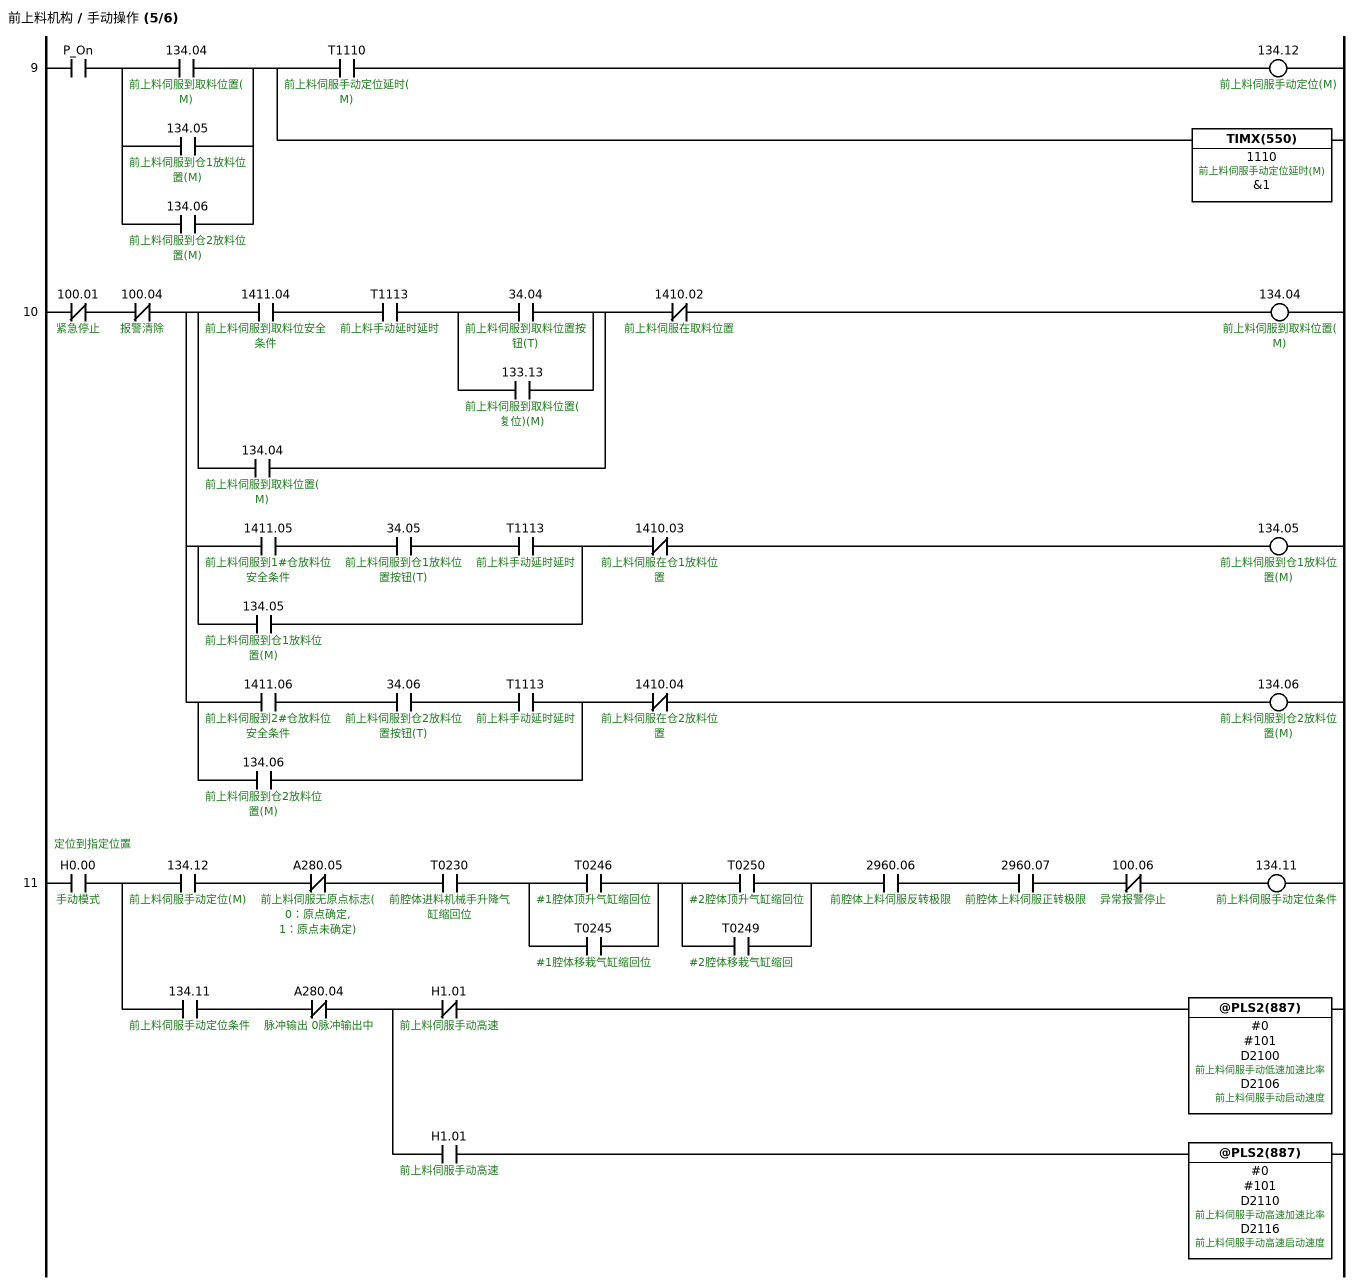
; rung 9
LD P_On
LD 134.04  ; 前上料伺服到取料位置(M)
OR 134.05  ; 前上料伺服到仓1放料位置(M)
OR 134.06  ; 前上料伺服到仓2放料位置(M)
ANDLD
OUT TR0
AND T1110  ; 前上料伺服手动定位延时(M)
OUT 134.12  ; 前上料伺服手动定位(M)
LD TR0
TIMX(550) 1110 &1  ; 前上料伺服手动定位延时(M)
; rung 10
LDNOT 100.01  ; 紧急停止
ANDNOT 100.04  ; 报警清除
OUT TR0
LD 1411.04  ; 前上料伺服到取料位安全条件
AND T1113  ; 前上料手动延时延时
LD 34.04  ; 前上料伺服到取料位置按钮(T)
OR 133.13  ; 前上料伺服到取料位置(复位)(M)
ANDLD
OR 134.04  ; 前上料伺服到取料位置(M)
ANDLD
ANDNOT 1410.02  ; 前上料伺服在取料位置
OUT 134.04  ; 前上料伺服到取料位置(M)
LD TR0
LD 1411.05  ; 前上料伺服到1#仓放料位安全条件
AND 34.05  ; 前上料伺服到仓1放料位置按钮(T)
AND T1113  ; 前上料手动延时延时
OR 134.05  ; 前上料伺服到仓1放料位置(M)
ANDLD
ANDNOT 1410.03  ; 前上料伺服在仓1放料位置
OUT 134.05  ; 前上料伺服到仓1放料位置(M)
LD TR0
LD 1411.06  ; 前上料伺服到2#仓放料位安全条件
AND 34.06  ; 前上料伺服到仓2放料位置按钮(T)
AND T1113  ; 前上料手动延时延时
OR 134.06  ; 前上料伺服到仓2放料位置(M)
ANDLD
ANDNOT 1410.04  ; 前上料伺服在仓2放料位置
OUT 134.06  ; 前上料伺服到仓2放料位置(M)
; rung 11: 定位到指定位置
LD H0.00  ; 手动模式
OUT TR0
AND 134.12  ; 前上料伺服手动定位(M)
ANDNOT A280.05  ; 前上料伺服无原点标志(0：原点确定,1：原点未确定)
AND T0230  ; 前腔体进料机械手升降气缸缩回位
LD T0246  ; #1腔体顶升气缸缩回位
OR T0245  ; #1腔体移栽气缸缩回位
ANDLD
LD T0250  ; #2腔体顶升气缸缩回位
OR T0249  ; #2腔体移栽气缸缩回
ANDLD
AND 2960.06  ; 前腔体上料伺服反转极限
AND 2960.07  ; 前腔体上料伺服正转极限
ANDNOT 100.06  ; 异常报警停止
OUT 134.11  ; 前上料伺服手动定位条件
LD TR0
AND 134.11  ; 前上料伺服手动定位条件
ANDNOT A280.04  ; 脉冲输出 0脉冲输出中
OUT TR0
ANDNOT H1.01  ; 前上料伺服手动高速
@PLS2(887) #0 #101 D2100 D2106  ; 前上料伺服手动低速加速比率, 前上料伺服手动启动速度
LD TR0
AND H1.01  ; 前上料伺服手动高速
@PLS2(887) #0 #101 D2110 D2116  ; 前上料伺服手动高速加速比率, 前上料伺服手动高速启动速度

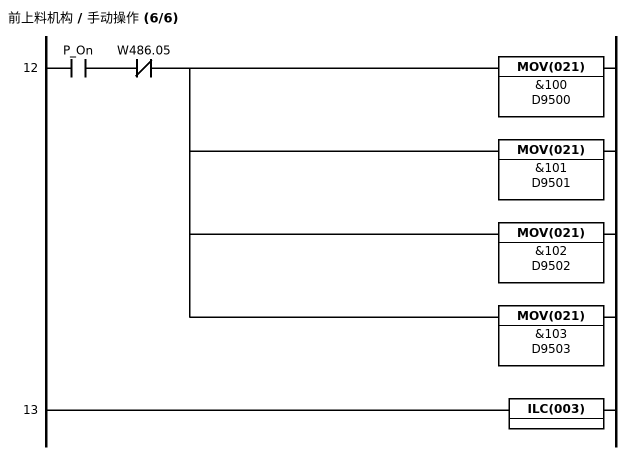
; rung 12
LD P_On
ANDNOT W486.05
MOV(021) &100 D9500
MOV(021) &101 D9501
MOV(021) &102 D9502
MOV(021) &103 D9503
; rung 13
ILC(003)

### Section 自动运行

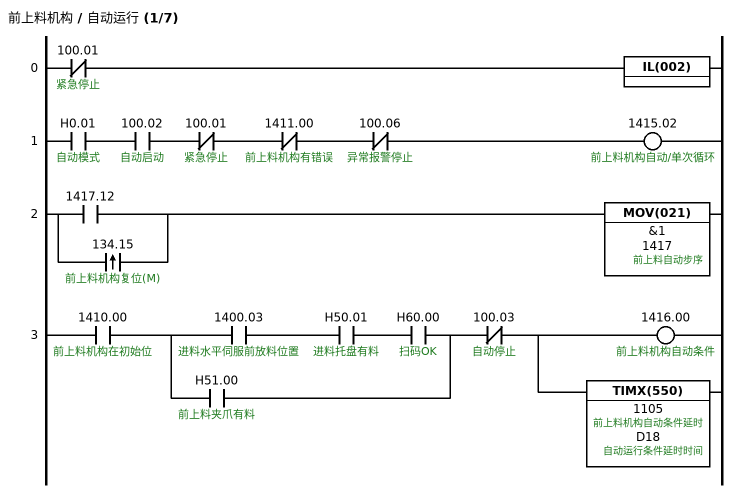
; rung 0
LDNOT 100.01  ; 紧急停止
IL(002)
; rung 1
LD H0.01  ; 自动模式
AND 100.02  ; 自动启动
ANDNOT 100.01  ; 紧急停止
ANDNOT 1411.00  ; 前上料机构有错误
ANDNOT 100.06  ; 异常报警停止
OUT 1415.02  ; 前上料机构自动/单次循环
; rung 2
LD 1417.12
@OR 134.15  ; 前上料机构复位(M)
MOV(021) &1 1417  ; 前上料自动步序
; rung 3
LD 1410.00  ; 前上料机构在初始位
LD 1400.03  ; 进料水平伺服前放料位置
AND H50.01  ; 进料托盘有料
AND H60.00  ; 扫码OK
OR H51.00  ; 前上料夹爪有料
ANDLD
ANDNOT 100.03  ; 自动停止
OUT 1416.00  ; 前上料机构自动条件
TIMX(550) 1105 D18  ; 自动运行条件延时时间, 前上料机构自动条件延时

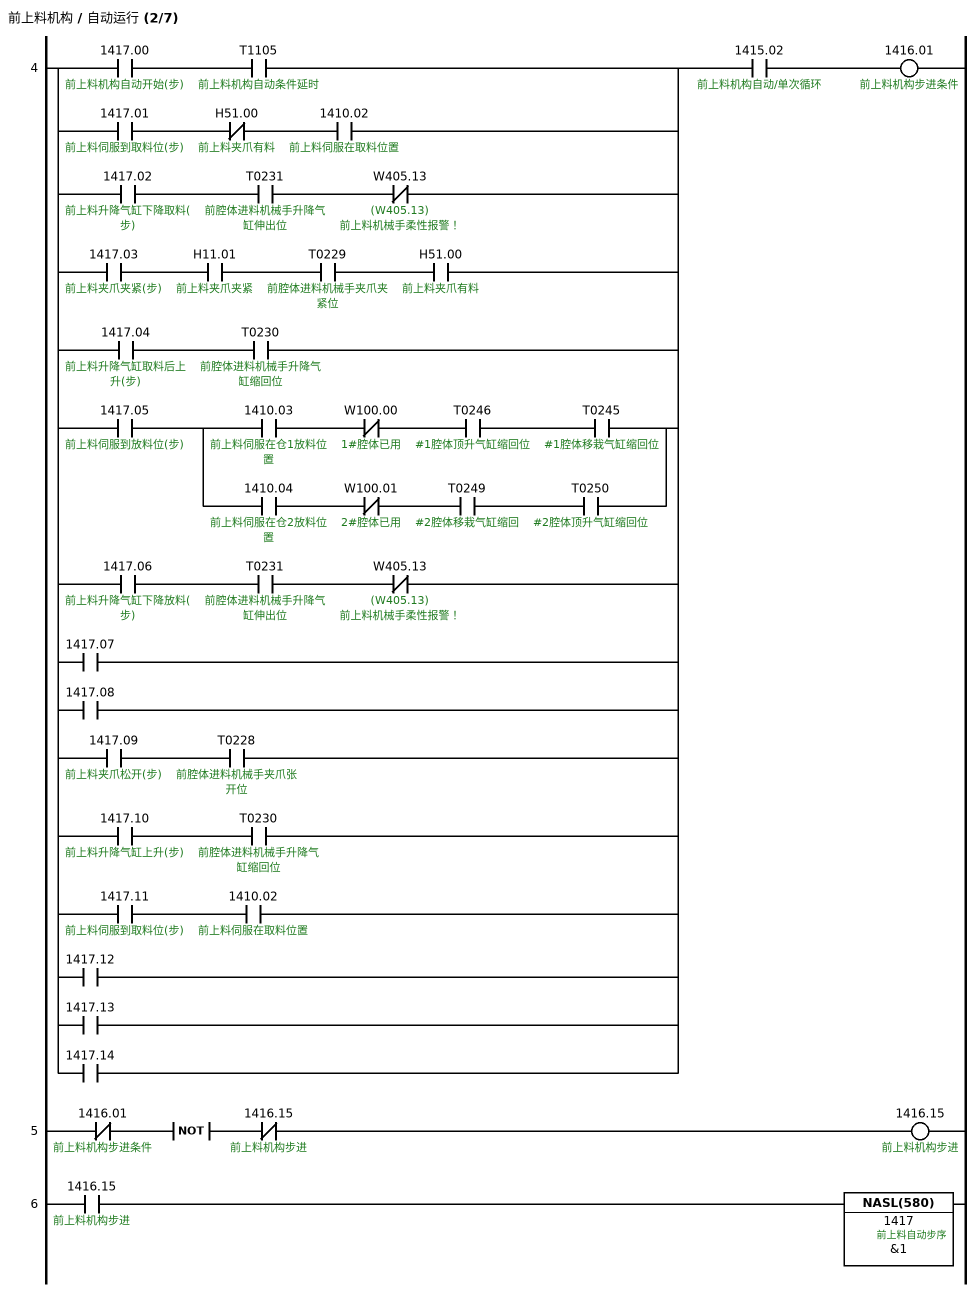
; rung 4
LD 1417.00  ; 前上料机构自动开始(步)
AND T1105  ; 前上料机构自动条件延时
LD 1417.01  ; 前上料伺服到取料位(步)
ANDNOT H51.00  ; 前上料夹爪有料
AND 1410.02  ; 前上料伺服在取料位置
ORLD
LD 1417.02  ; 前上料升降气缸下降取料(步)
AND T0231  ; 前腔体进料机械手升降气缸伸出位
ANDNOT W405.13  ; (W405.13) 前上料机械手柔性报警！
ORLD
LD 1417.03  ; 前上料夹爪夹紧(步)
AND H11.01  ; 前上料夹爪夹紧
AND T0229  ; 前腔体进料机械手夹爪夹紧位
AND H51.00  ; 前上料夹爪有料
ORLD
LD 1417.04  ; 前上料升降气缸取料后上升(步)
AND T0230  ; 前腔体进料机械手升降气缸缩回位
ORLD
LD 1417.05  ; 前上料伺服到放料位(步)
LD 1410.03  ; 前上料伺服在仓1放料位置
ANDNOT W100.00  ; 1#腔体已用
AND T0246  ; #1腔体顶升气缸缩回位
AND T0245  ; #1腔体移栽气缸缩回位
LD 1410.04  ; 前上料伺服在仓2放料位置
ANDNOT W100.01  ; 2#腔体已用
AND T0249  ; #2腔体移栽气缸缩回
AND T0250  ; #2腔体顶升气缸缩回位
ORLD
ANDLD
ORLD
LD 1417.06  ; 前上料升降气缸下降放料(步)
AND T0231  ; 前腔体进料机械手升降气缸伸出位
ANDNOT W405.13  ; (W405.13) 前上料机械手柔性报警！
ORLD
OR 1417.07
OR 1417.08
LD 1417.09  ; 前上料夹爪松开(步)
AND T0228  ; 前腔体进料机械手夹爪张开位
ORLD
LD 1417.10  ; 前上料升降气缸上升(步)
AND T0230  ; 前腔体进料机械手升降气缸缩回位
ORLD
LD 1417.11  ; 前上料伺服到取料位(步)
AND 1410.02  ; 前上料伺服在取料位置
ORLD
OR 1417.12
OR 1417.13
OR 1417.14
AND 1415.02  ; 前上料机构自动/单次循环
OUT 1416.01  ; 前上料机构步进条件
; rung 5
LDNOT 1416.01  ; 前上料机构步进条件
NOT(520)
ANDNOT 1416.15  ; 前上料机构步进
OUT 1416.15  ; 前上料机构步进
; rung 6
LD 1416.15  ; 前上料机构步进
NASL(580) 1417 &1  ; 前上料自动步序

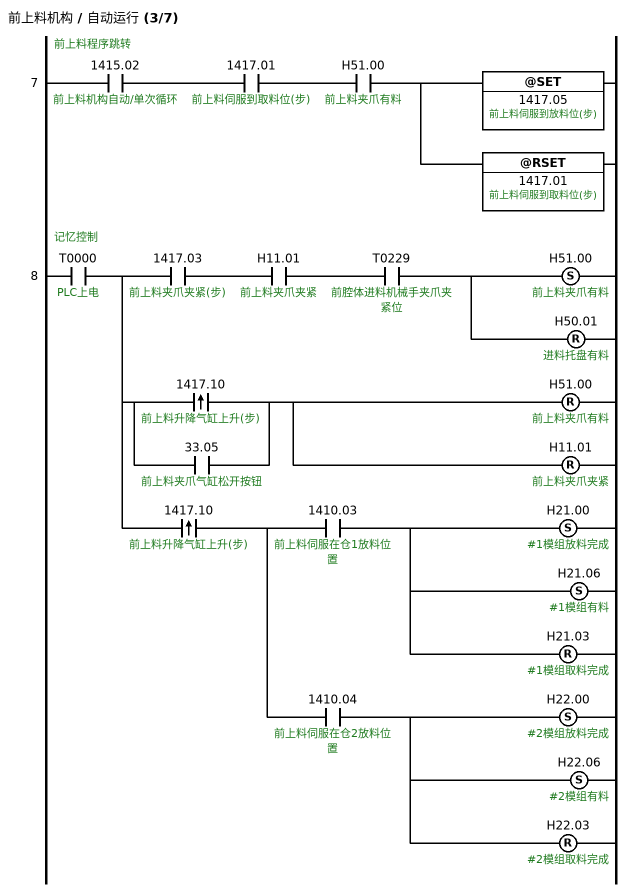
; rung 7: 前上料程序跳转
LD 1415.02  ; 前上料机构自动/单次循环
AND 1417.01  ; 前上料伺服到取料位(步)
AND H51.00  ; 前上料夹爪有料
@SET 1417.05  ; 前上料伺服到放料位(步)
@RSET 1417.01  ; 前上料伺服到取料位(步)
; rung 8: 记忆控制
LD T0000  ; PLC上电
OUT TR0
AND 1417.03  ; 前上料夹爪夹紧(步)
AND H11.01  ; 前上料夹爪夹紧
AND T0229  ; 前腔体进料机械手夹爪夹紧位
SET H51.00  ; 前上料夹爪有料
RSET H50.01  ; 进料托盘有料
LD TR0
@LD 1417.10  ; 前上料升降气缸上升(步)
OR 33.05  ; 前上料夹爪气缸松开按钮
ANDLD
RSET H51.00  ; 前上料夹爪有料
RSET H11.01  ; 前上料夹爪夹紧
LD TR0
@AND 1417.10  ; 前上料升降气缸上升(步)
OUT TR0
AND 1410.03  ; 前上料伺服在仓1放料位置
SET H21.00  ; #1模组放料完成
SET H21.06  ; #1模组有料
RSET H21.03  ; #1模组取料完成
LD TR0
AND 1410.04  ; 前上料伺服在仓2放料位置
SET H22.00  ; #2模组放料完成
SET H22.06  ; #2模组有料
RSET H22.03  ; #2模组取料完成

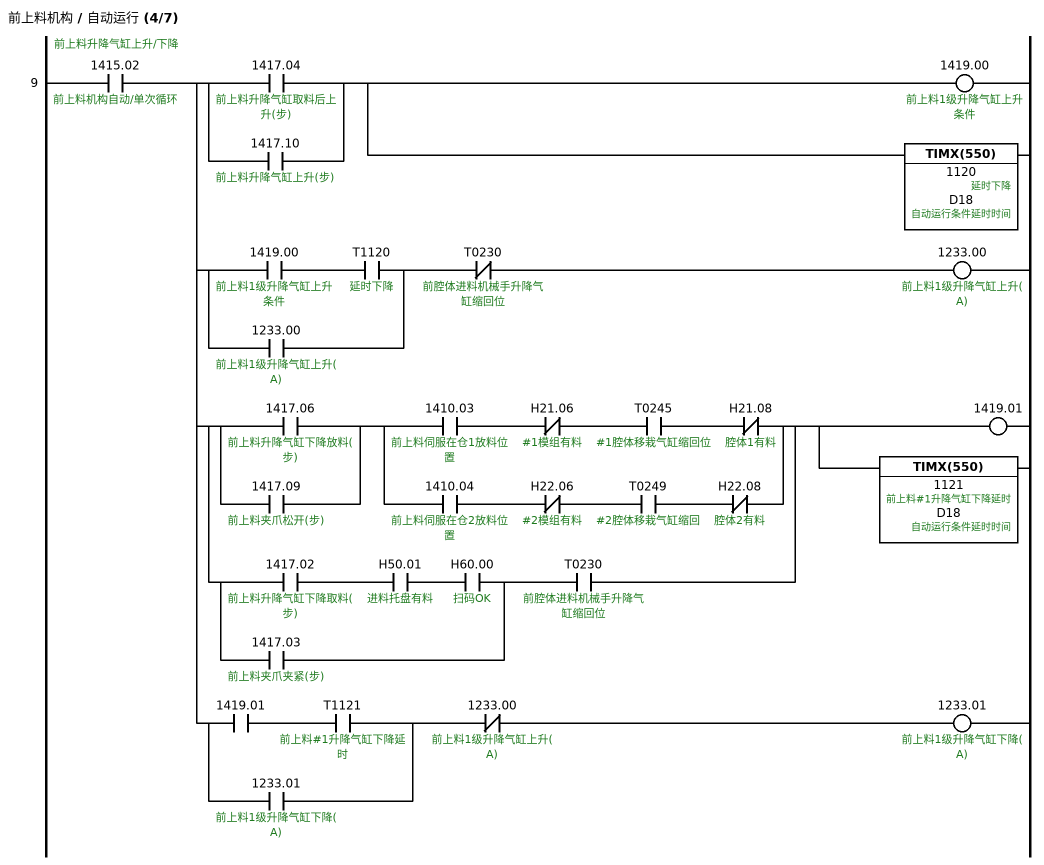
; rung 9: 前上料升降气缸上升/下降
LD 1415.02  ; 前上料机构自动/单次循环
OUT TR0
LD 1417.04  ; 前上料升降气缸取料后上升(步)
OR 1417.10  ; 前上料升降气缸上升(步)
ANDLD
OUT 1419.00  ; 前上料1级升降气缸上升条件
TIMX(550) 1120 D18  ; 自动运行条件延时时间, 延时下降
LD TR0
LD 1419.00  ; 前上料1级升降气缸上升条件
AND T1120  ; 延时下降
OR 1233.00  ; 前上料1级升降气缸上升(A)
ANDLD
ANDNOT T0230  ; 前腔体进料机械手升降气缸缩回位
OUT 1233.00  ; 前上料1级升降气缸上升(A)
LD TR0
LD 1417.06  ; 前上料升降气缸下降放料(步)
OR 1417.09  ; 前上料夹爪松开(步)
LD 1410.03  ; 前上料伺服在仓1放料位置
ANDNOT H21.06  ; #1模组有料
AND T0245  ; #1腔体移栽气缸缩回位
ANDNOT H21.08  ; 腔体1有料
LD 1410.04  ; 前上料伺服在仓2放料位置
ANDNOT H22.06  ; #2模组有料
AND T0249  ; #2腔体移栽气缸缩回
ANDNOT H22.08  ; 腔体2有料
ORLD
ANDLD
LD 1417.02  ; 前上料升降气缸下降取料(步)
AND H50.01  ; 进料托盘有料
AND H60.00  ; 扫码OK
OR 1417.03  ; 前上料夹爪夹紧(步)
AND T0230  ; 前腔体进料机械手升降气缸缩回位
ORLD
ANDLD
OUT 1419.01
TIMX(550) 1121 D18  ; 自动运行条件延时时间, 前上料#1升降气缸下降延时
LD TR0
LD 1419.01
AND T1121  ; 前上料#1升降气缸下降延时
OR 1233.01  ; 前上料1级升降气缸下降(A)
ANDLD
ANDNOT 1233.00  ; 前上料1级升降气缸上升(A)
OUT 1233.01  ; 前上料1级升降气缸下降(A)

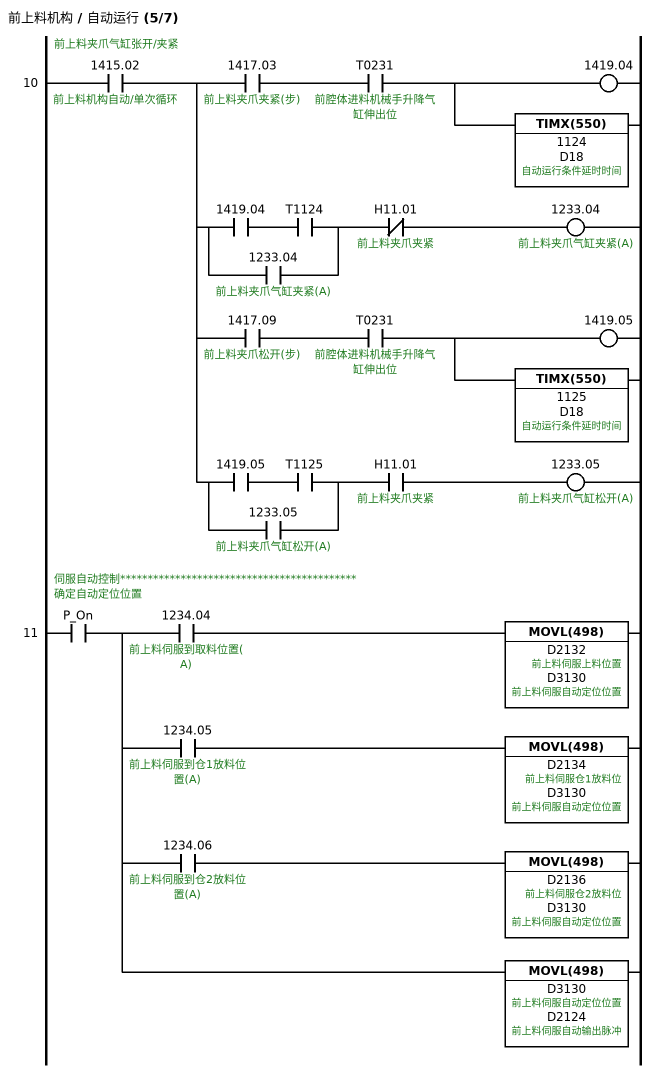
; rung 10: 前上料夹爪气缸张开/夹紧
LD 1415.02  ; 前上料机构自动/单次循环
OUT TR0
AND 1417.03  ; 前上料夹爪夹紧(步)
AND T0231  ; 前腔体进料机械手升降气缸伸出位
OUT 1419.04
TIMX(550) 1124 D18  ; 自动运行条件延时时间
LD TR0
LD 1419.04
AND T1124
OR 1233.04  ; 前上料夹爪气缸夹紧(A)
ANDLD
ANDNOT H11.01  ; 前上料夹爪夹紧
OUT 1233.04  ; 前上料夹爪气缸夹紧(A)
LD TR0
AND 1417.09  ; 前上料夹爪松开(步)
AND T0231  ; 前腔体进料机械手升降气缸伸出位
OUT 1419.05
TIMX(550) 1125 D18  ; 自动运行条件延时时间
LD TR0
LD 1419.05
AND T1125
OR 1233.05  ; 前上料夹爪气缸松开(A)
ANDLD
AND H11.01  ; 前上料夹爪夹紧
OUT 1233.05  ; 前上料夹爪气缸松开(A)
; rung 11: 伺服自动控制******************************************* / 确定自动定位位置
LD P_On
OUT TR0
AND 1234.04  ; 前上料伺服到取料位置(A)
MOVL(498) D2132 D3130  ; 前上料伺服上料位置, 前上料伺服自动定位位置
LD TR0
AND 1234.05  ; 前上料伺服到仓1放料位置(A)
MOVL(498) D2134 D3130  ; 前上料伺服仓1放料位, 前上料伺服自动定位位置
LD TR0
AND 1234.06  ; 前上料伺服到仓2放料位置(A)
MOVL(498) D2136 D3130  ; 前上料伺服仓2放料位, 前上料伺服自动定位位置
LD TR0
MOVL(498) D3130 D2124  ; 前上料伺服自动定位位置, 前上料伺服自动输出脉冲

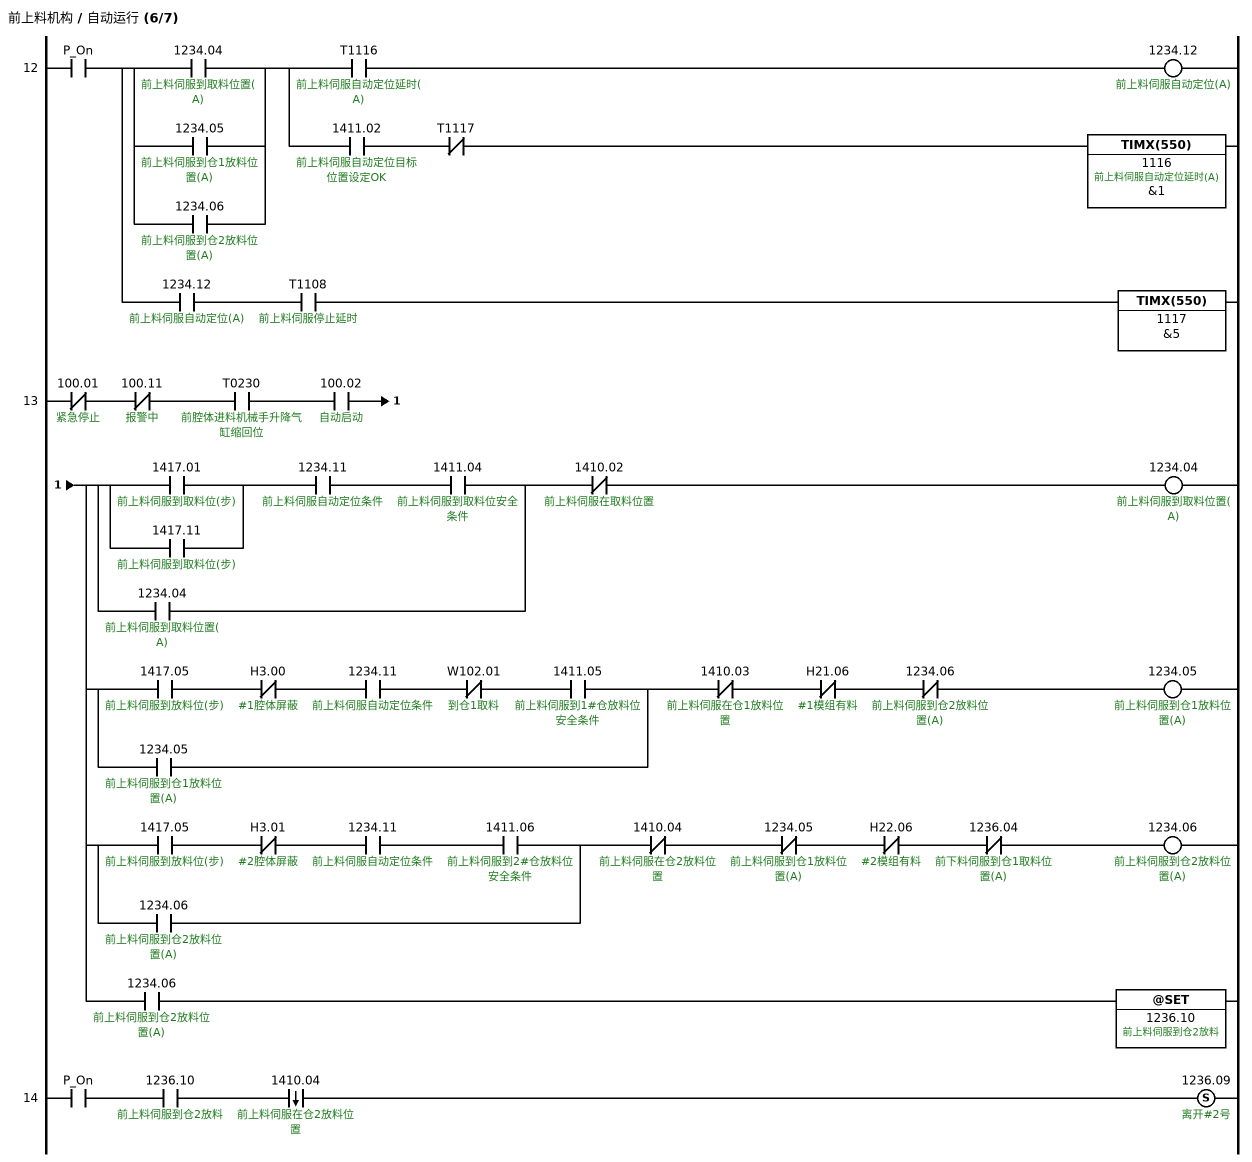
; rung 12
LD P_On
OUT TR0
LD 1234.04  ; 前上料伺服到取料位置(A)
OR 1234.05  ; 前上料伺服到仓1放料位置(A)
OR 1234.06  ; 前上料伺服到仓2放料位置(A)
ANDLD
OUT TR1
AND T1116  ; 前上料伺服自动定位延时(A)
OUT 1234.12  ; 前上料伺服自动定位(A)
LD TR1
AND 1411.02  ; 前上料伺服自动定位目标位置设定OK
ANDNOT T1117
TIMX(550) 1116 &1  ; 前上料伺服自动定位延时(A)
LD TR0
AND 1234.12  ; 前上料伺服自动定位(A)
AND T1108  ; 前上料伺服停止延时
TIMX(550) 1117 &5
; rung 13
LDNOT 100.01  ; 紧急停止
ANDNOT 100.11  ; 报警中
AND T0230  ; 前腔体进料机械手升降气缸缩回位
AND 100.02  ; 自动启动
OUT TR0
LD 1417.01  ; 前上料伺服到取料位(步)
OR 1417.11  ; 前上料伺服到取料位(步)
AND 1234.11  ; 前上料伺服自动定位条件
AND 1411.04  ; 前上料伺服到取料位安全条件
OR 1234.04  ; 前上料伺服到取料位置(A)
ANDLD
ANDNOT 1410.02  ; 前上料伺服在取料位置
OUT 1234.04  ; 前上料伺服到取料位置(A)
LD TR0
LD 1417.05  ; 前上料伺服到放料位(步)
ANDNOT H3.00  ; #1腔体屏蔽
AND 1234.11  ; 前上料伺服自动定位条件
ANDNOT W102.01  ; 到仓1取料
AND 1411.05  ; 前上料伺服到1#仓放料位安全条件
OR 1234.05  ; 前上料伺服到仓1放料位置(A)
ANDLD
ANDNOT 1410.03  ; 前上料伺服在仓1放料位置
ANDNOT H21.06  ; #1模组有料
ANDNOT 1234.06  ; 前上料伺服到仓2放料位置(A)
OUT 1234.05  ; 前上料伺服到仓1放料位置(A)
LD TR0
LD 1417.05  ; 前上料伺服到放料位(步)
ANDNOT H3.01  ; #2腔体屏蔽
AND 1234.11  ; 前上料伺服自动定位条件
AND 1411.06  ; 前上料伺服到2#仓放料位安全条件
OR 1234.06  ; 前上料伺服到仓2放料位置(A)
ANDLD
ANDNOT 1410.04  ; 前上料伺服在仓2放料位置
ANDNOT 1234.05  ; 前上料伺服到仓1放料位置(A)
ANDNOT H22.06  ; #2模组有料
ANDNOT 1236.04  ; 前下料伺服到仓1取料位置(A)
OUT 1234.06  ; 前上料伺服到仓2放料位置(A)
LD TR0
AND 1234.06  ; 前上料伺服到仓2放料位置(A)
@SET 1236.10  ; 前上料伺服到仓2放料
; rung 14
LD P_On
AND 1236.10  ; 前上料伺服到仓2放料
%AND 1410.04  ; 前上料伺服在仓2放料位置
SET 1236.09  ; 离开#2号

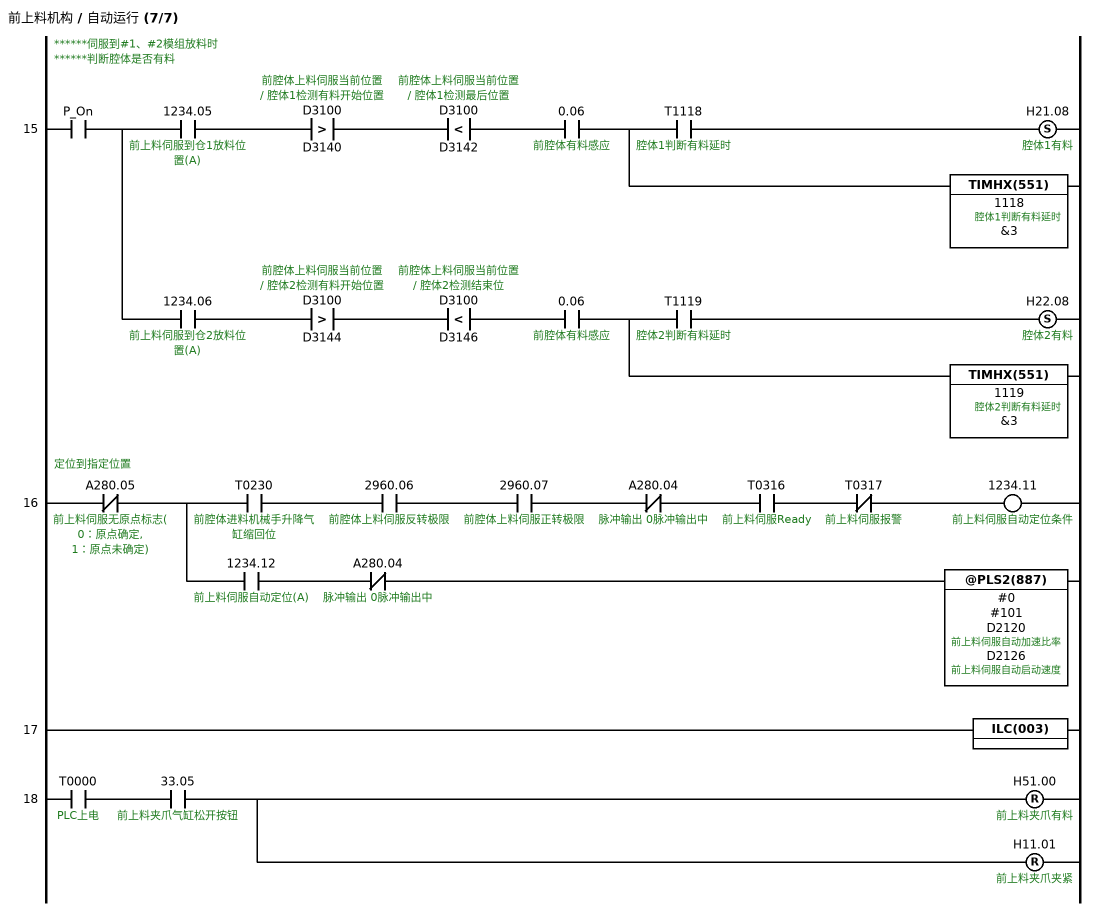
; rung 15: ******伺服到#1、#2模组放料时 / ******判断腔体是否有料
LD P_On
OUT TR0
AND 1234.05  ; 前上料伺服到仓1放料位置(A)
AND>SL(323) D3100 D3140  ; 前腔体上料伺服当前位置, 腔体1检测有料开始位置
AND<SL(313) D3100 D3142  ; 前腔体上料伺服当前位置, 腔体1检测最后位置
AND 0.06  ; 前腔体有料感应
OUT TR1
AND T1118  ; 腔体1判断有料延时
SET H21.08  ; 腔体1有料
LD TR1
TIMHX(551) 1118 &3  ; 腔体1判断有料延时
LD TR0
AND 1234.06  ; 前上料伺服到仓2放料位置(A)
AND>SL(323) D3100 D3144  ; 前腔体上料伺服当前位置, 腔体2检测有料开始位置
AND<SL(313) D3100 D3146  ; 前腔体上料伺服当前位置, 腔体2检测结束位
AND 0.06  ; 前腔体有料感应
OUT TR0
AND T1119  ; 腔体2判断有料延时
SET H22.08  ; 腔体2有料
LD TR0
TIMHX(551) 1119 &3  ; 腔体2判断有料延时
; rung 16: 定位到指定位置
LDNOT A280.05  ; 前上料伺服无原点标志(0：原点确定,1：原点未确定)
OUT TR0
AND T0230  ; 前腔体进料机械手升降气缸缩回位
AND 2960.06  ; 前腔体上料伺服反转极限
AND 2960.07  ; 前腔体上料伺服正转极限
ANDNOT A280.04  ; 脉冲输出 0脉冲输出中
AND T0316  ; 前上料伺服Ready
ANDNOT T0317  ; 前上料伺服报警
OUT 1234.11  ; 前上料伺服自动定位条件
LD TR0
AND 1234.12  ; 前上料伺服自动定位(A)
ANDNOT A280.04  ; 脉冲输出 0脉冲输出中
@PLS2(887) #0 #101 D2120 D2126  ; 前上料伺服自动加速比率, 前上料伺服自动启动速度
; rung 17
ILC(003)
; rung 18
LD T0000  ; PLC上电
AND 33.05  ; 前上料夹爪气缸松开按钮
RSET H51.00  ; 前上料夹爪有料
RSET H11.01  ; 前上料夹爪夹紧

### Section 外部输出

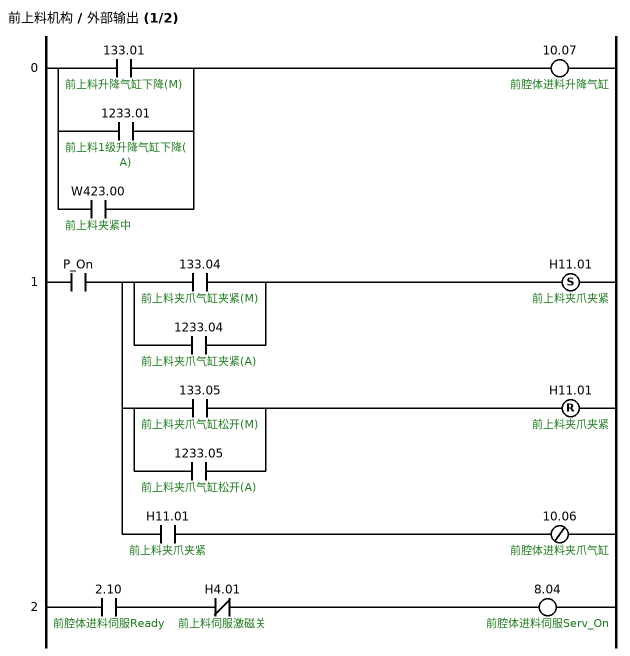
; rung 0
LD 133.01  ; 前上料升降气缸下降(M)
OR 1233.01  ; 前上料1级升降气缸下降(A)
OR W423.00  ; 前上料夹紧中
OUT 10.07  ; 前腔体进料升降气缸
; rung 1
LD P_On
OUT TR0
LD 133.04  ; 前上料夹爪气缸夹紧(M)
OR 1233.04  ; 前上料夹爪气缸夹紧(A)
ANDLD
SET H11.01  ; 前上料夹爪夹紧
LD TR0
LD 133.05  ; 前上料夹爪气缸松开(M)
OR 1233.05  ; 前上料夹爪气缸松开(A)
ANDLD
RSET H11.01  ; 前上料夹爪夹紧
LD TR0
AND H11.01  ; 前上料夹爪夹紧
OUTNOT 10.06  ; 前腔体进料夹爪气缸
; rung 2
LD 2.10  ; 前腔体进料伺服Ready
ANDNOT H4.01  ; 前上料伺服激磁关
OUT 8.04  ; 前腔体进料伺服Serv_On

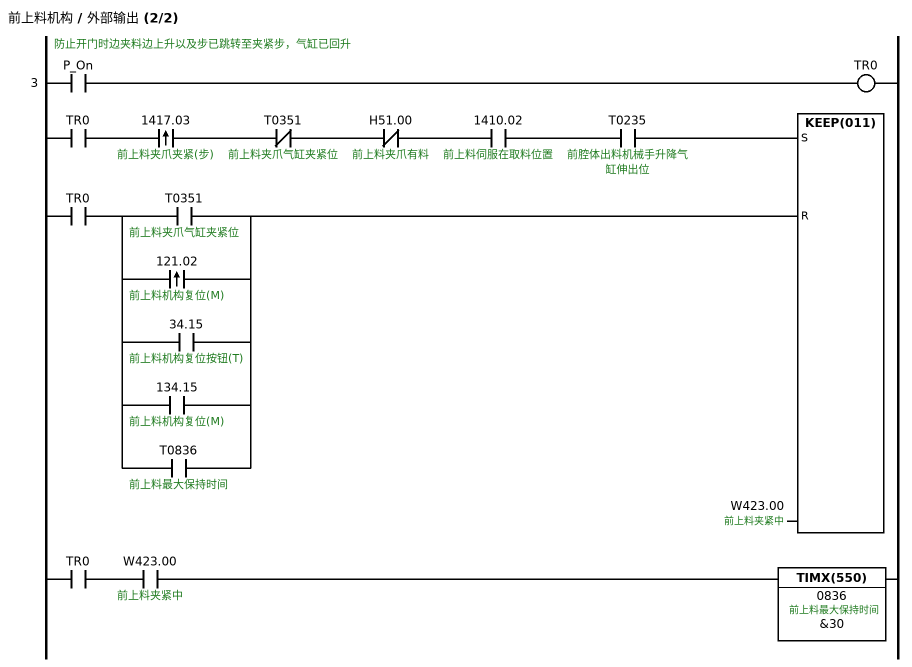
; rung 3: 防止开门时边夹料边上升以及步已跳转至夹紧步，气缸已回升
LD P_On
OUT TR0
@AND 1417.03  ; 前上料夹爪夹紧(步)
ANDNOT T0351  ; 前上料夹爪气缸夹紧位
ANDNOT H51.00  ; 前上料夹爪有料
AND 1410.02  ; 前上料伺服在取料位置
AND T0235  ; 前腔体出料机械手升降气缸伸出位
LD TR0
LD T0351  ; 前上料夹爪气缸夹紧位
@OR 121.02  ; 前上料机构复位(M)
OR 34.15  ; 前上料机构复位按钮(T)
OR 134.15  ; 前上料机构复位(M)
OR T0836  ; 前上料最大保持时间
ANDLD
KEEP(011) W423.00  ; 前上料夹紧中
LD TR0
AND W423.00  ; 前上料夹紧中
TIMX(550) 0836 &30  ; 前上料最大保持时间

### Section 指示灯
; rung 0: ************************************************** / 气缸动作及位置指示灯

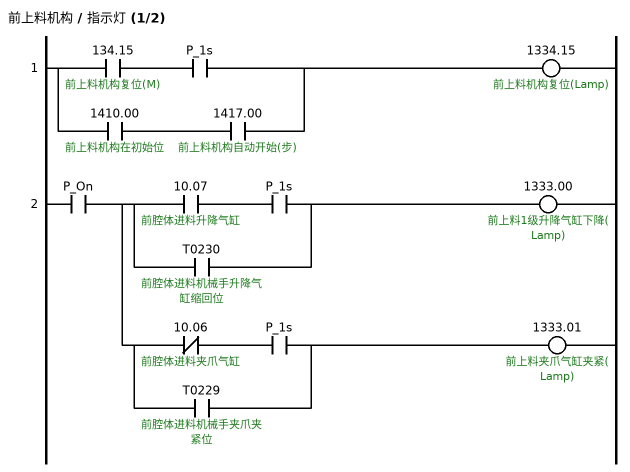
; rung 1
LD 134.15  ; 前上料机构复位(M)
AND P_1s
LD 1410.00  ; 前上料机构在初始位
AND 1417.00  ; 前上料机构自动开始(步)
ORLD
OUT 1334.15  ; 前上料机构复位(Lamp)
; rung 2
LD P_On
OUT TR0
LD 10.07  ; 前腔体进料升降气缸
AND P_1s
OR T0230  ; 前腔体进料机械手升降气缸缩回位
ANDLD
OUT 1333.00  ; 前上料1级升降气缸下降(Lamp)
LD TR0
LDNOT 10.06  ; 前腔体进料夹爪气缸
AND P_1s
OR T0229  ; 前腔体进料机械手夹爪夹紧位
ANDLD
OUT 1333.01  ; 前上料夹爪气缸夹紧(Lamp)

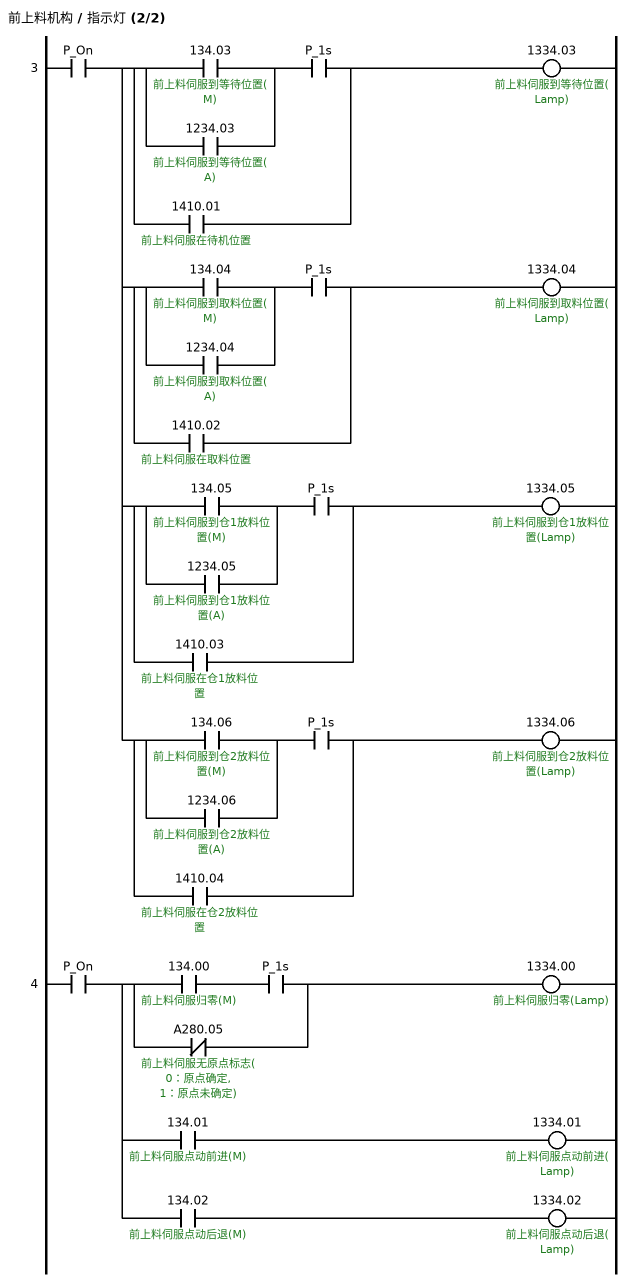
; rung 3
LD P_On
OUT TR0
LD 134.03  ; 前上料伺服到等待位置(M)
OR 1234.03  ; 前上料伺服到等待位置(A)
AND P_1s
OR 1410.01  ; 前上料伺服在待机位置
ANDLD
OUT 1334.03  ; 前上料伺服到等待位置(Lamp)
LD TR0
LD 134.04  ; 前上料伺服到取料位置(M)
OR 1234.04  ; 前上料伺服到取料位置(A)
AND P_1s
OR 1410.02  ; 前上料伺服在取料位置
ANDLD
OUT 1334.04  ; 前上料伺服到取料位置(Lamp)
LD TR0
LD 134.05  ; 前上料伺服到仓1放料位置(M)
OR 1234.05  ; 前上料伺服到仓1放料位置(A)
AND P_1s
OR 1410.03  ; 前上料伺服在仓1放料位置
ANDLD
OUT 1334.05  ; 前上料伺服到仓1放料位置(Lamp)
LD TR0
LD 134.06  ; 前上料伺服到仓2放料位置(M)
OR 1234.06  ; 前上料伺服到仓2放料位置(A)
AND P_1s
OR 1410.04  ; 前上料伺服在仓2放料位置
ANDLD
OUT 1334.06  ; 前上料伺服到仓2放料位置(Lamp)
; rung 4
LD P_On
OUT TR0
LD 134.00  ; 前上料伺服归零(M)
AND P_1s
ORNOT A280.05  ; 前上料伺服无原点标志(0：原点确定,1：原点未确定)
ANDLD
OUT 1334.00  ; 前上料伺服归零(Lamp)
LD TR0
AND 134.01  ; 前上料伺服点动前进(M)
OUT 1334.01  ; 前上料伺服点动前进(Lamp)
LD TR0
AND 134.02  ; 前上料伺服点动后退(M)
OUT 1334.02  ; 前上料伺服点动后退(Lamp)

### Section END
; rung 0
END(001)

## Program 前下料机构 (cyclic task 3)

### Section Main

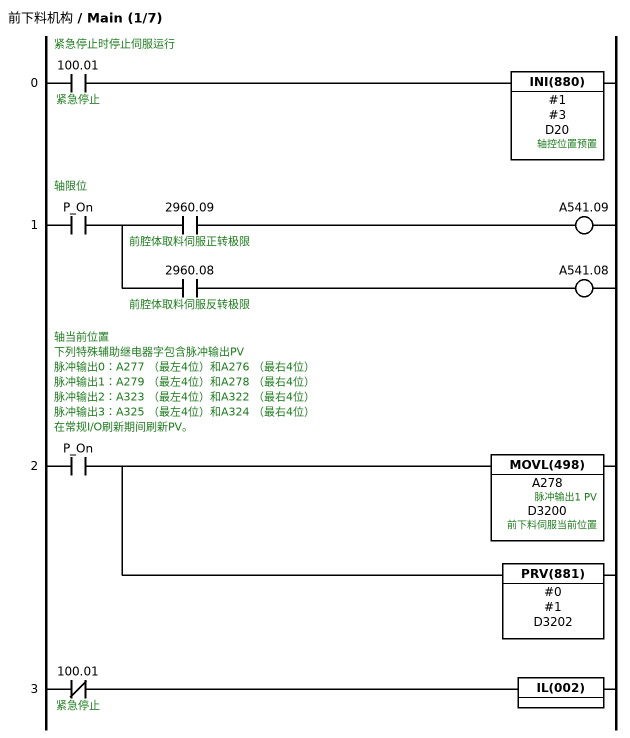
; rung 0: 紧急停止时停止伺服运行
LD 100.01  ; 紧急停止
INI(880) #1 #3 D20  ; 轴控位置预置
; rung 1: 轴限位
LD P_On
OUT TR0
AND 2960.09  ; 前腔体取料伺服正转极限
OUT A541.09
LD TR0
AND 2960.08  ; 前腔体取料伺服反转极限
OUT A541.08
; rung 2: 轴当前位置 / 下列特殊辅助继电器字包含脉冲输出PV / 脉冲输出0：A277 （最左4位）和A276 （最右4位） / 脉冲输出1：A279 （最左4位）和A278 （最右4位） / 脉冲输出2：A323 （最左4位）和A322 （最右4位） / 脉冲输出3：A325 （最左4位）和A324 （最右4位） / 在常规I/O刷新期间刷新PV。
LD P_On
MOVL(498) A278 D3200  ; 脉冲输出1 PV, 前下料伺服当前位置
PRV(881) #0 #1 D3202
; rung 3
LDNOT 100.01  ; 紧急停止
IL(002)

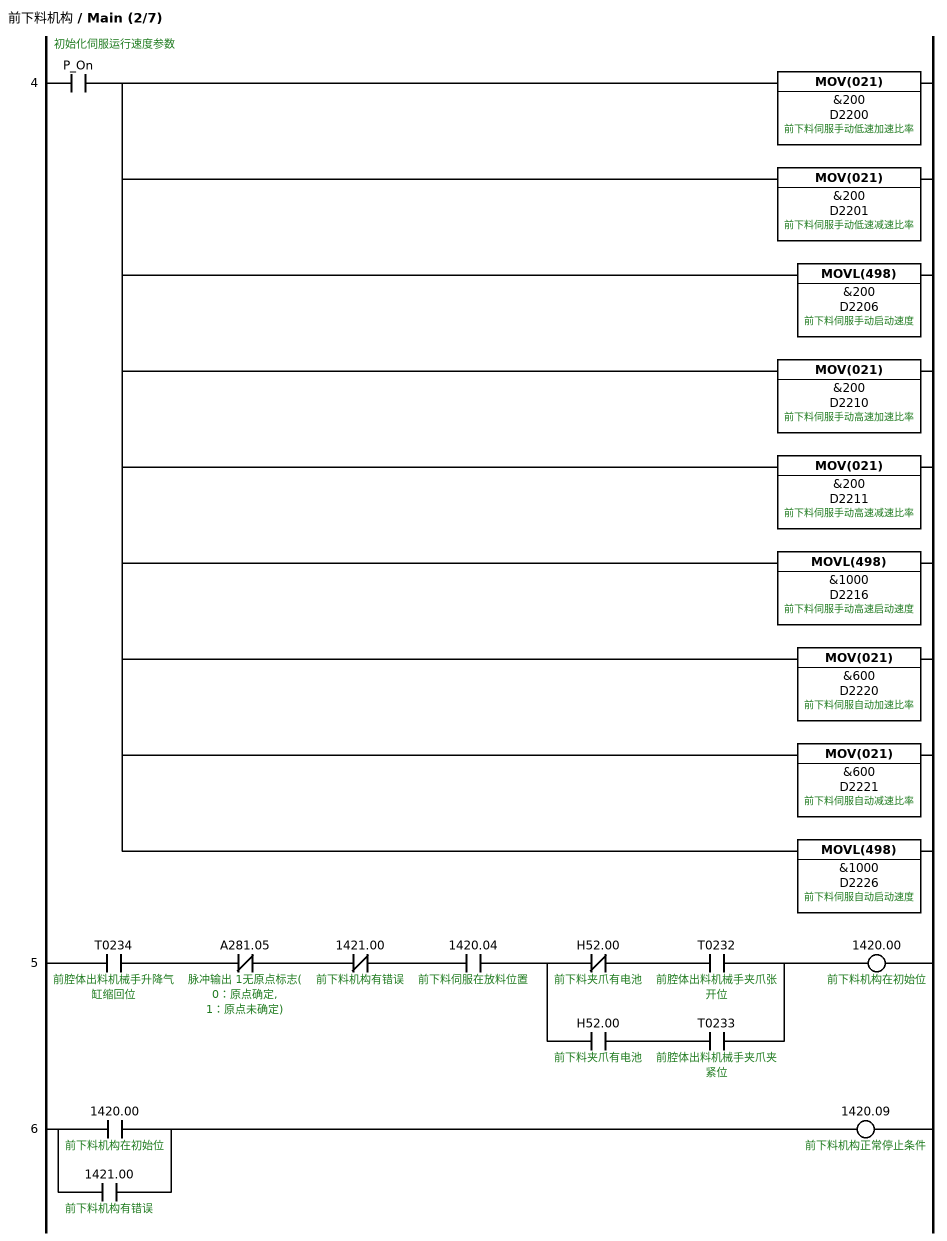
; rung 4: 初始化伺服运行速度参数
LD P_On
MOV(021) &200 D2200  ; 前下料伺服手动低速加速比率
MOV(021) &200 D2201  ; 前下料伺服手动低速减速比率
MOVL(498) &200 D2206  ; 前下料伺服手动启动速度
MOV(021) &200 D2210  ; 前下料伺服手动高速加速比率
MOV(021) &200 D2211  ; 前下料伺服手动高速减速比率
MOVL(498) &1000 D2216  ; 前下料伺服手动高速启动速度
MOV(021) &600 D2220  ; 前下料伺服自动加速比率
MOV(021) &600 D2221  ; 前下料伺服自动减速比率
MOVL(498) &1000 D2226  ; 前下料伺服自动启动速度
; rung 5
LD T0234  ; 前腔体出料机械手升降气缸缩回位
ANDNOT A281.05  ; 脉冲输出 1无原点标志(0：原点确定,1：原点未确定)
ANDNOT 1421.00  ; 前下料机构有错误
AND 1420.04  ; 前下料伺服在放料位置
LDNOT H52.00  ; 前下料夹爪有电池
AND T0232  ; 前腔体出料机械手夹爪张开位
LD H52.00  ; 前下料夹爪有电池
AND T0233  ; 前腔体出料机械手夹爪夹紧位
ORLD
ANDLD
OUT 1420.00  ; 前下料机构在初始位
; rung 6
LD 1420.00  ; 前下料机构在初始位
OR 1421.00  ; 前下料机构有错误
OUT 1420.09  ; 前下料机构正常停止条件

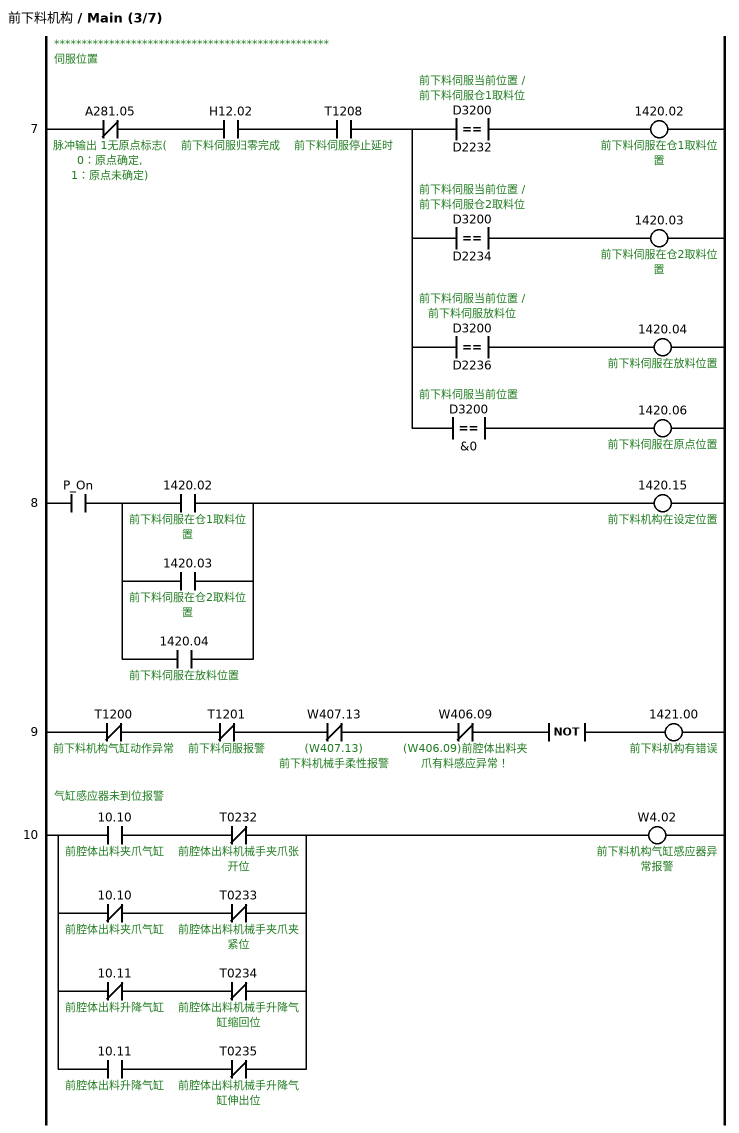
; rung 7: ************************************************** / 伺服位置
LDNOT A281.05  ; 脉冲输出 1无原点标志(0：原点确定,1：原点未确定)
AND H12.02  ; 前下料伺服归零完成
AND T1208  ; 前下料伺服停止延时
OUT TR0
AND=SL(303) D3200 D2232  ; 前下料伺服当前位置, 前下料伺服仓1取料位
OUT 1420.02  ; 前下料伺服在仓1取料位置
LD TR0
AND=SL(303) D3200 D2234  ; 前下料伺服当前位置, 前下料伺服仓2取料位
OUT 1420.03  ; 前下料伺服在仓2取料位置
LD TR0
AND=SL(303) D3200 D2236  ; 前下料伺服当前位置, 前下料伺服放料位
OUT 1420.04  ; 前下料伺服在放料位置
LD TR0
AND=SL(303) D3200 &0  ; 前下料伺服当前位置
OUT 1420.06  ; 前下料伺服在原点位置
; rung 8
LD P_On
LD 1420.02  ; 前下料伺服在仓1取料位置
OR 1420.03  ; 前下料伺服在仓2取料位置
OR 1420.04  ; 前下料伺服在放料位置
ANDLD
OUT 1420.15  ; 前下料机构在设定位置
; rung 9
LDNOT T1200  ; 前下料机构气缸动作异常
ANDNOT T1201  ; 前下料伺服报警
ANDNOT W407.13  ; (W407.13) 前下料机械手柔性报警
ANDNOT W406.09  ; (W406.09)前腔体出料夹爪有料感应异常！
NOT(520)
OUT 1421.00  ; 前下料机构有错误
; rung 10: 气缸感应器未到位报警
LD 10.10  ; 前腔体出料夹爪气缸
ANDNOT T0232  ; 前腔体出料机械手夹爪张开位
LDNOT 10.10  ; 前腔体出料夹爪气缸
ANDNOT T0233  ; 前腔体出料机械手夹爪夹紧位
ORLD
LDNOT 10.11  ; 前腔体出料升降气缸
ANDNOT T0234  ; 前腔体出料机械手升降气缸缩回位
ORLD
LD 10.11  ; 前腔体出料升降气缸
ANDNOT T0235  ; 前腔体出料机械手升降气缸伸出位
ORLD
OUT W4.02  ; 前下料机构气缸感应器异常报警

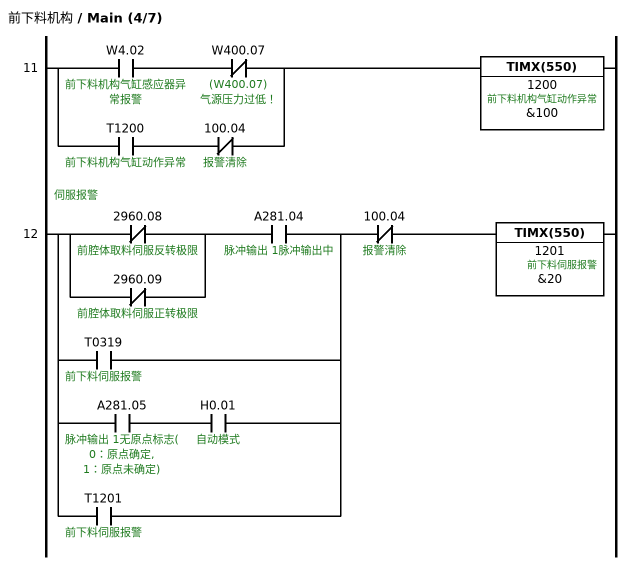
; rung 11
LD W4.02  ; 前下料机构气缸感应器异常报警
ANDNOT W400.07  ; (W400.07) 气源压力过低！
LD T1200  ; 前下料机构气缸动作异常
ANDNOT 100.04  ; 报警清除
ORLD
TIMX(550) 1200 &100  ; 前下料机构气缸动作异常
; rung 12: 伺服报警
LDNOT 2960.08  ; 前腔体取料伺服反转极限
ORNOT 2960.09  ; 前腔体取料伺服正转极限
AND A281.04  ; 脉冲输出 1脉冲输出中
OR T0319  ; 前下料伺服报警
LD A281.05  ; 脉冲输出 1无原点标志(0：原点确定,1：原点未确定)
AND H0.01  ; 自动模式
ORLD
OR T1201  ; 前下料伺服报警
ANDNOT 100.04  ; 报警清除
TIMX(550) 1201 &20  ; 前下料伺服报警

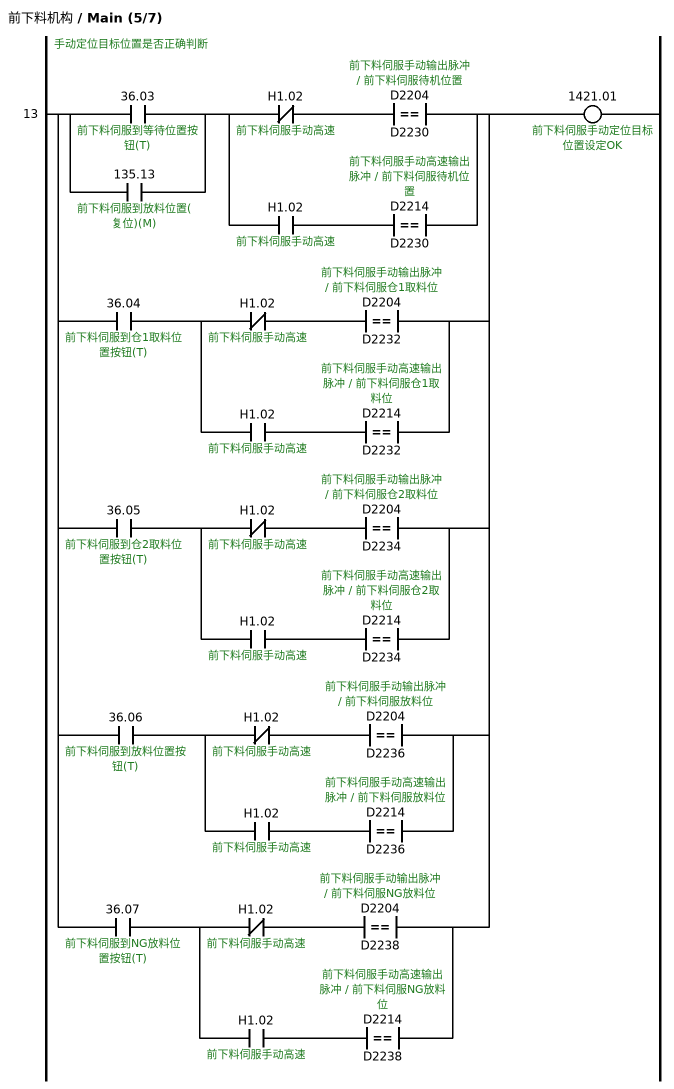
; rung 13: 手动定位目标位置是否正确判断
LD 36.03  ; 前下料伺服到等待位置按钮(T)
OR 135.13  ; 前下料伺服到放料位置(复位)(M)
LDNOT H1.02  ; 前下料伺服手动高速
AND=SL(303) D2204 D2230  ; 前下料伺服手动输出脉冲, 前下料伺服待机位置
LD H1.02  ; 前下料伺服手动高速
AND=SL(303) D2214 D2230  ; 前下料伺服手动高速输出脉冲, 前下料伺服待机位置
ORLD
ANDLD
LD 36.04  ; 前下料伺服到仓1取料位置按钮(T)
LDNOT H1.02  ; 前下料伺服手动高速
AND=SL(303) D2204 D2232  ; 前下料伺服手动输出脉冲, 前下料伺服仓1取料位
LD H1.02  ; 前下料伺服手动高速
AND=SL(303) D2214 D2232  ; 前下料伺服手动高速输出脉冲, 前下料伺服仓1取料位
ORLD
ANDLD
ORLD
LD 36.05  ; 前下料伺服到仓2取料位置按钮(T)
LDNOT H1.02  ; 前下料伺服手动高速
AND=SL(303) D2204 D2234  ; 前下料伺服手动输出脉冲, 前下料伺服仓2取料位
LD H1.02  ; 前下料伺服手动高速
AND=SL(303) D2214 D2234  ; 前下料伺服手动高速输出脉冲, 前下料伺服仓2取料位
ORLD
ANDLD
ORLD
LD 36.06  ; 前下料伺服到放料位置按钮(T)
LDNOT H1.02  ; 前下料伺服手动高速
AND=SL(303) D2204 D2236  ; 前下料伺服手动输出脉冲, 前下料伺服放料位
LD H1.02  ; 前下料伺服手动高速
AND=SL(303) D2214 D2236  ; 前下料伺服手动高速输出脉冲, 前下料伺服放料位
ORLD
ANDLD
ORLD
LD 36.07  ; 前下料伺服到NG放料位置按钮(T)
LDNOT H1.02  ; 前下料伺服手动高速
AND=SL(303) D2204 D2238  ; 前下料伺服手动输出脉冲, 前下料伺服NG放料位
LD H1.02  ; 前下料伺服手动高速
AND=SL(303) D2214 D2238  ; 前下料伺服手动高速输出脉冲, 前下料伺服NG放料位
ORLD
ANDLD
ORLD
OUT 1421.01  ; 前下料伺服手动定位目标位置设定OK

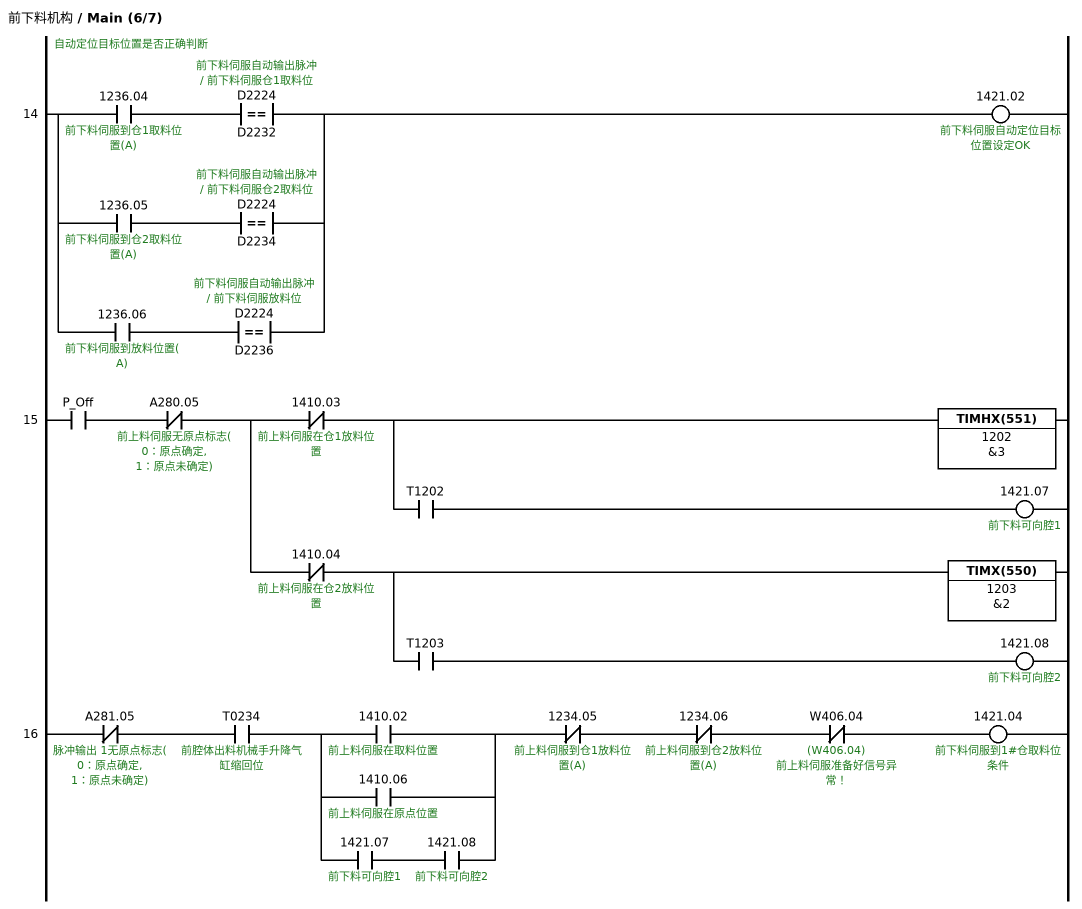
; rung 14: 自动定位目标位置是否正确判断
LD 1236.04  ; 前下料伺服到仓1取料位置(A)
AND=SL(303) D2224 D2232  ; 前下料伺服自动输出脉冲, 前下料伺服仓1取料位
LD 1236.05  ; 前下料伺服到仓2取料位置(A)
AND=SL(303) D2224 D2234  ; 前下料伺服自动输出脉冲, 前下料伺服仓2取料位
ORLD
LD 1236.06  ; 前下料伺服到放料位置(A)
AND=SL(303) D2224 D2236  ; 前下料伺服自动输出脉冲, 前下料伺服放料位
ORLD
OUT 1421.02  ; 前下料伺服自动定位目标位置设定OK
; rung 15
LD P_Off
ANDNOT A280.05  ; 前上料伺服无原点标志(0：原点确定,1：原点未确定)
OUT TR0
ANDNOT 1410.03  ; 前上料伺服在仓1放料位置
TIMHX(551) 1202 &3
AND T1202
OUT 1421.07  ; 前下料可向腔1
LD TR0
ANDNOT 1410.04  ; 前上料伺服在仓2放料位置
TIMX(550) 1203 &2
AND T1203
OUT 1421.08  ; 前下料可向腔2
; rung 16
LDNOT A281.05  ; 脉冲输出 1无原点标志(0：原点确定,1：原点未确定)
AND T0234  ; 前腔体出料机械手升降气缸缩回位
LD 1410.02  ; 前上料伺服在取料位置
OR 1410.06  ; 前上料伺服在原点位置
LD 1421.07  ; 前下料可向腔1
AND 1421.08  ; 前下料可向腔2
ORLD
ANDLD
ANDNOT 1234.05  ; 前上料伺服到仓1放料位置(A)
ANDNOT 1234.06  ; 前上料伺服到仓2放料位置(A)
ANDNOT W406.04  ; (W406.04) 前上料伺服准备好信号异常！
OUT 1421.04  ; 前下料伺服到1#仓取料位条件

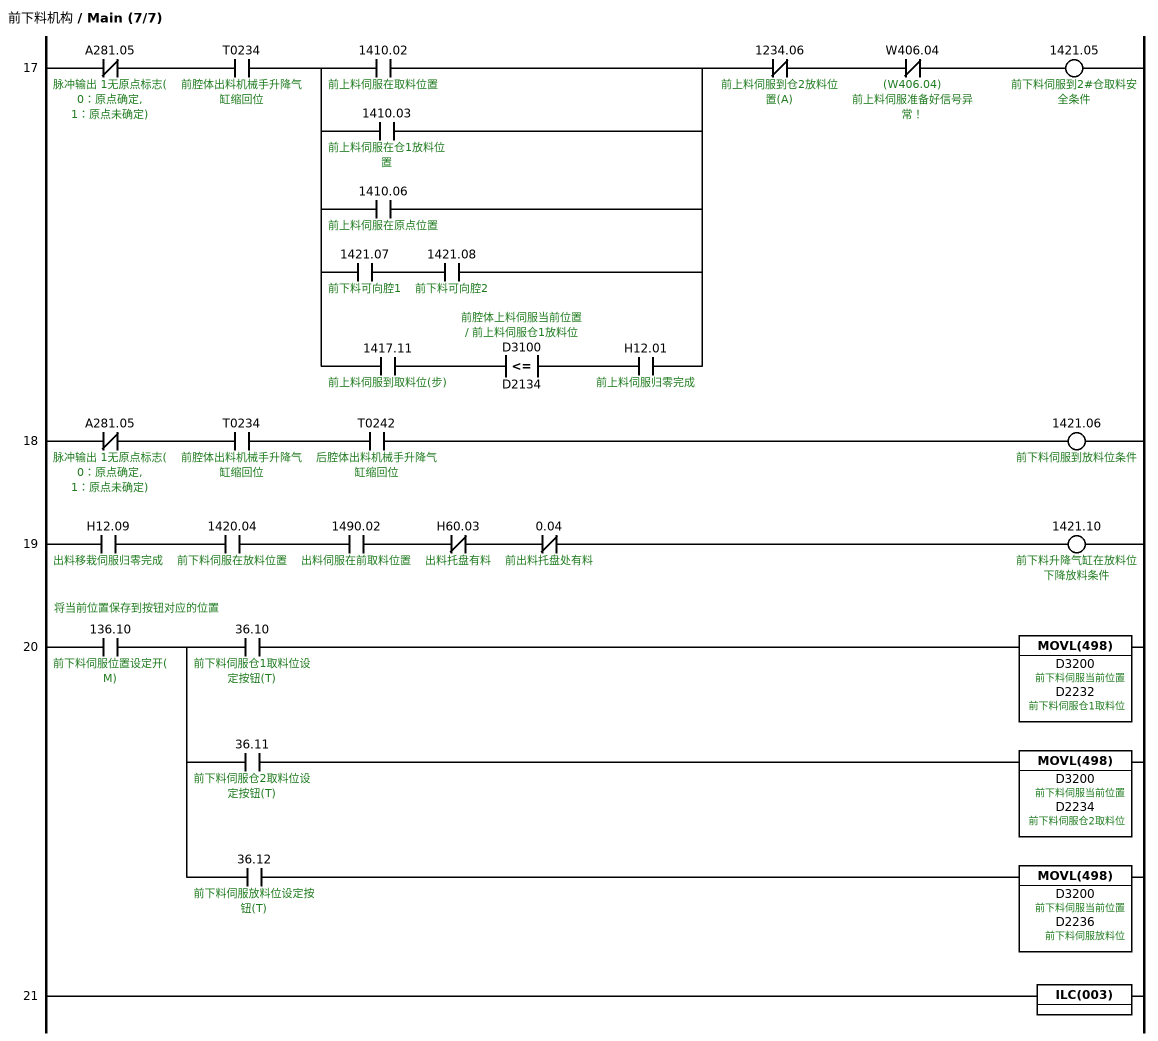
; rung 17
LDNOT A281.05  ; 脉冲输出 1无原点标志(0：原点确定,1：原点未确定)
AND T0234  ; 前腔体出料机械手升降气缸缩回位
LD 1410.02  ; 前上料伺服在取料位置
OR 1410.03  ; 前上料伺服在仓1放料位置
OR 1410.06  ; 前上料伺服在原点位置
LD 1421.07  ; 前下料可向腔1
AND 1421.08  ; 前下料可向腔2
ORLD
LD 1417.11  ; 前上料伺服到取料位(步)
AND<=SL(318) D3100 D2134  ; 前腔体上料伺服当前位置, 前上料伺服仓1放料位
AND H12.01  ; 前上料伺服归零完成
ORLD
ANDLD
ANDNOT 1234.06  ; 前上料伺服到仓2放料位置(A)
ANDNOT W406.04  ; (W406.04) 前上料伺服准备好信号异常！
OUT 1421.05  ; 前下料伺服到2#仓取料安全条件
; rung 18
LDNOT A281.05  ; 脉冲输出 1无原点标志(0：原点确定,1：原点未确定)
AND T0234  ; 前腔体出料机械手升降气缸缩回位
AND T0242  ; 后腔体出料机械手升降气缸缩回位
OUT 1421.06  ; 前下料伺服到放料位条件
; rung 19
LD H12.09  ; 出料移栽伺服归零完成
AND 1420.04  ; 前下料伺服在放料位置
AND 1490.02  ; 出料伺服在前取料位置
ANDNOT H60.03  ; 出料托盘有料
ANDNOT 0.04  ; 前出料托盘处有料
OUT 1421.10  ; 前下料升降气缸在放料位下降放料条件
; rung 20: 将当前位置保存到按钮对应的位置
LD 136.10  ; 前下料伺服位置设定开(M)
OUT TR0
AND 36.10  ; 前下料伺服仓1取料位设定按钮(T)
MOVL(498) D3200 D2232  ; 前下料伺服当前位置, 前下料伺服仓1取料位
LD TR0
AND 36.11  ; 前下料伺服仓2取料位设定按钮(T)
MOVL(498) D3200 D2234  ; 前下料伺服当前位置, 前下料伺服仓2取料位
LD TR0
AND 36.12  ; 前下料伺服放料位设定按钮(T)
MOVL(498) D3200 D2236  ; 前下料伺服当前位置, 前下料伺服放料位
; rung 21
ILC(003)

### Section 工站复位

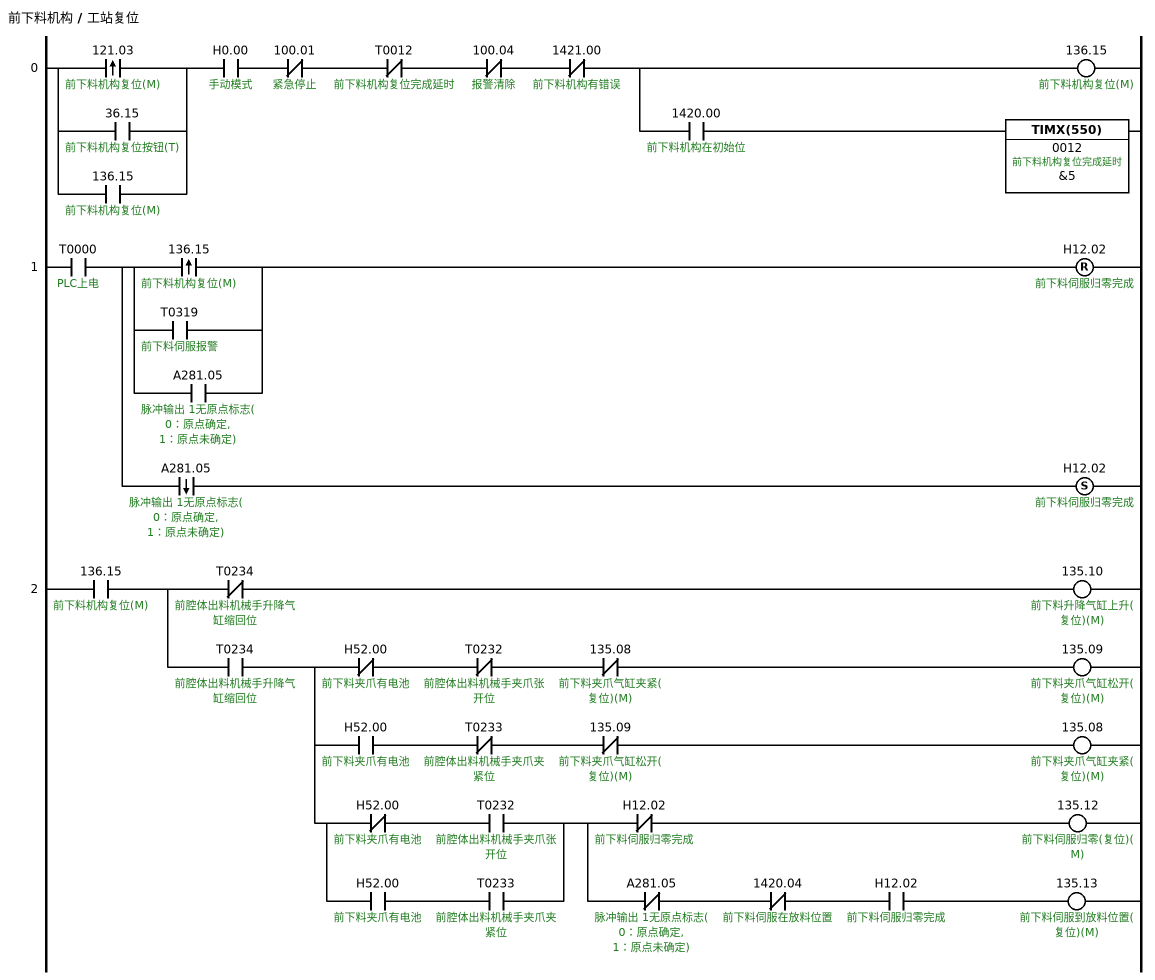
; rung 0
@LD 121.03  ; 前下料机构复位(M)
OR 36.15  ; 前下料机构复位按钮(T)
OR 136.15  ; 前下料机构复位(M)
AND H0.00  ; 手动模式
ANDNOT 100.01  ; 紧急停止
ANDNOT T0012  ; 前下料机构复位完成延时
ANDNOT 100.04  ; 报警清除
ANDNOT 1421.00  ; 前下料机构有错误
OUT 136.15  ; 前下料机构复位(M)
AND 1420.00  ; 前下料机构在初始位
TIMX(550) 0012 &5  ; 前下料机构复位完成延时
; rung 1
LD T0000  ; PLC上电
OUT TR0
@LD 136.15  ; 前下料机构复位(M)
OR T0319  ; 前下料伺服报警
OR A281.05  ; 脉冲输出 1无原点标志(0：原点确定,1：原点未确定)
ANDLD
RSET H12.02  ; 前下料伺服归零完成
LD TR0
%AND A281.05  ; 脉冲输出 1无原点标志(0：原点确定,1：原点未确定)
SET H12.02  ; 前下料伺服归零完成
; rung 2
LD 136.15  ; 前下料机构复位(M)
OUT TR0
ANDNOT T0234  ; 前腔体出料机械手升降气缸缩回位
OUT 135.10  ; 前下料升降气缸上升(复位)(M)
LD TR0
AND T0234  ; 前腔体出料机械手升降气缸缩回位
OUT TR0
ANDNOT H52.00  ; 前下料夹爪有电池
ANDNOT T0232  ; 前腔体出料机械手夹爪张开位
ANDNOT 135.08  ; 前下料夹爪气缸夹紧(复位)(M)
OUT 135.09  ; 前下料夹爪气缸松开(复位)(M)
LD TR0
AND H52.00  ; 前下料夹爪有电池
ANDNOT T0233  ; 前腔体出料机械手夹爪夹紧位
ANDNOT 135.09  ; 前下料夹爪气缸松开(复位)(M)
OUT 135.08  ; 前下料夹爪气缸夹紧(复位)(M)
LD TR0
LDNOT H52.00  ; 前下料夹爪有电池
AND T0232  ; 前腔体出料机械手夹爪张开位
LD H52.00  ; 前下料夹爪有电池
AND T0233  ; 前腔体出料机械手夹爪夹紧位
ORLD
ANDLD
OUT TR0
ANDNOT H12.02  ; 前下料伺服归零完成
OUT 135.12  ; 前下料伺服归零(复位)(M)
LD TR0
ANDNOT A281.05  ; 脉冲输出 1无原点标志(0：原点确定,1：原点未确定)
ANDNOT 1420.04  ; 前下料伺服在放料位置
AND H12.02  ; 前下料伺服归零完成
OUT 135.13  ; 前下料伺服到放料位置(复位)(M)

### Section 手动操作

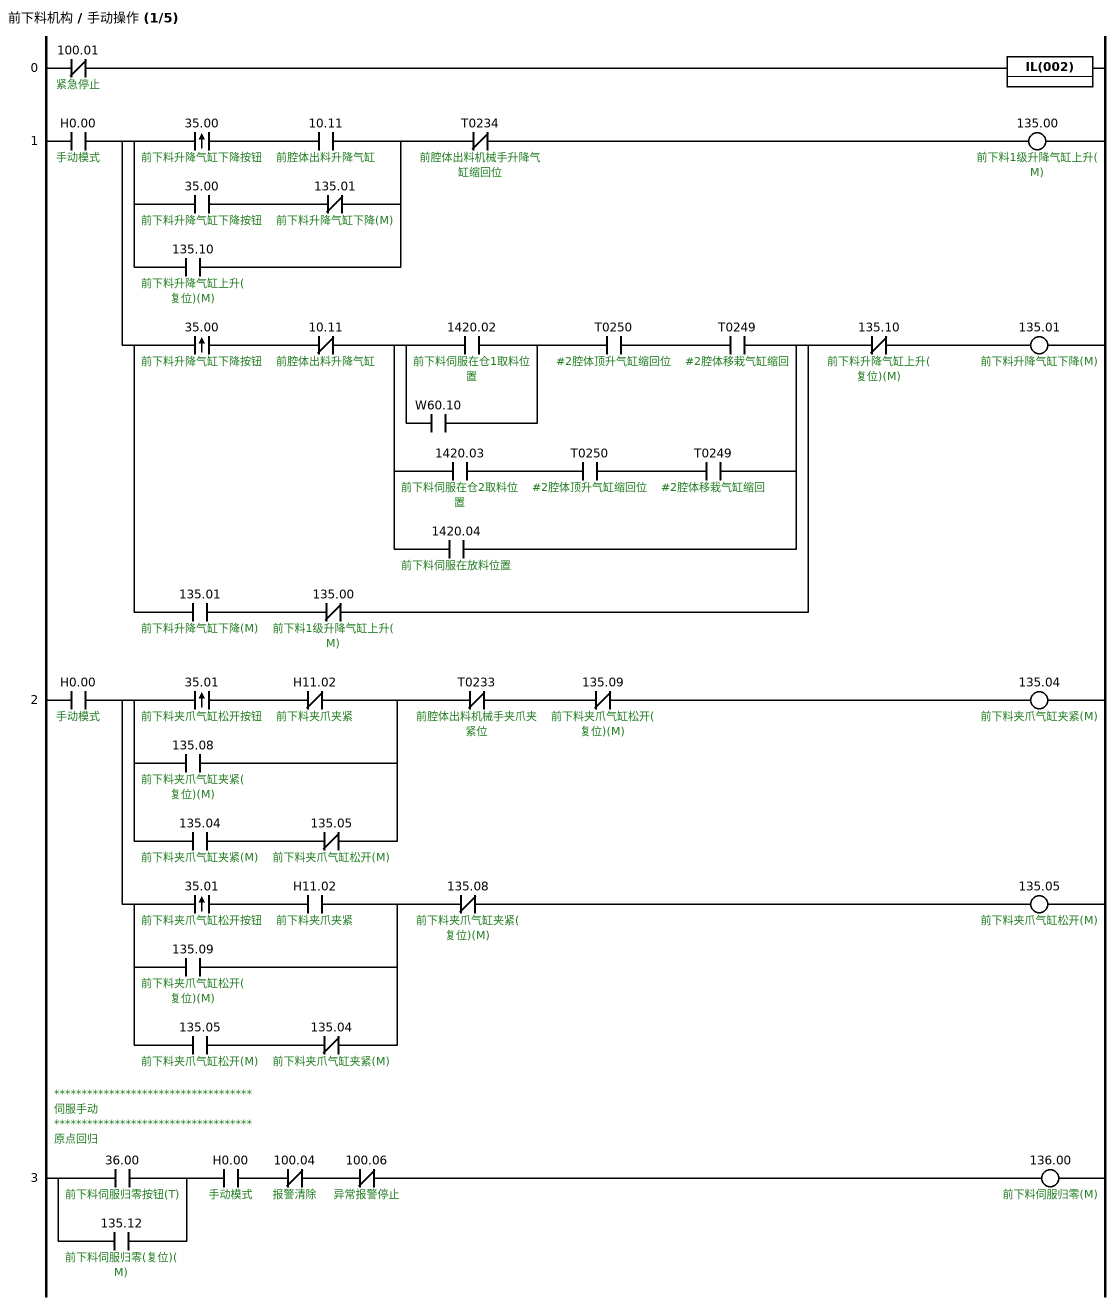
; rung 0
LDNOT 100.01  ; 紧急停止
IL(002)
; rung 1
LD H0.00  ; 手动模式
OUT TR0
@LD 35.00  ; 前下料升降气缸下降按钮
AND 10.11  ; 前腔体出料升降气缸
LD 35.00  ; 前下料升降气缸下降按钮
ANDNOT 135.01  ; 前下料升降气缸下降(M)
ORLD
OR 135.10  ; 前下料升降气缸上升(复位)(M)
ANDLD
ANDNOT T0234  ; 前腔体出料机械手升降气缸缩回位
OUT 135.00  ; 前下料1级升降气缸上升(M)
LD TR0
@LD 35.00  ; 前下料升降气缸下降按钮
ANDNOT 10.11  ; 前腔体出料升降气缸
LD 1420.02  ; 前下料伺服在仓1取料位置
OR W60.10
AND T0250  ; #2腔体顶升气缸缩回位
AND T0249  ; #2腔体移栽气缸缩回
LD 1420.03  ; 前下料伺服在仓2取料位置
AND T0250  ; #2腔体顶升气缸缩回位
AND T0249  ; #2腔体移栽气缸缩回
ORLD
OR 1420.04  ; 前下料伺服在放料位置
ANDLD
LD 135.01  ; 前下料升降气缸下降(M)
ANDNOT 135.00  ; 前下料1级升降气缸上升(M)
ORLD
ANDLD
ANDNOT 135.10  ; 前下料升降气缸上升(复位)(M)
OUT 135.01  ; 前下料升降气缸下降(M)
; rung 2
LD H0.00  ; 手动模式
OUT TR0
@LD 35.01  ; 前下料夹爪气缸松开按钮
ANDNOT H11.02  ; 前下料夹爪夹紧
OR 135.08  ; 前下料夹爪气缸夹紧(复位)(M)
LD 135.04  ; 前下料夹爪气缸夹紧(M)
ANDNOT 135.05  ; 前下料夹爪气缸松开(M)
ORLD
ANDLD
ANDNOT T0233  ; 前腔体出料机械手夹爪夹紧位
ANDNOT 135.09  ; 前下料夹爪气缸松开(复位)(M)
OUT 135.04  ; 前下料夹爪气缸夹紧(M)
LD TR0
@LD 35.01  ; 前下料夹爪气缸松开按钮
AND H11.02  ; 前下料夹爪夹紧
OR 135.09  ; 前下料夹爪气缸松开(复位)(M)
LD 135.05  ; 前下料夹爪气缸松开(M)
ANDNOT 135.04  ; 前下料夹爪气缸夹紧(M)
ORLD
ANDLD
ANDNOT 135.08  ; 前下料夹爪气缸夹紧(复位)(M)
OUT 135.05  ; 前下料夹爪气缸松开(M)
; rung 3: ************************************ / 伺服手动 / ************************************ / 原点回归
LD 36.00  ; 前下料伺服归零按钮(T)
OR 135.12  ; 前下料伺服归零(复位)(M)
AND H0.00  ; 手动模式
ANDNOT 100.04  ; 报警清除
ANDNOT 100.06  ; 异常报警停止
OUT 136.00  ; 前下料伺服归零(M)

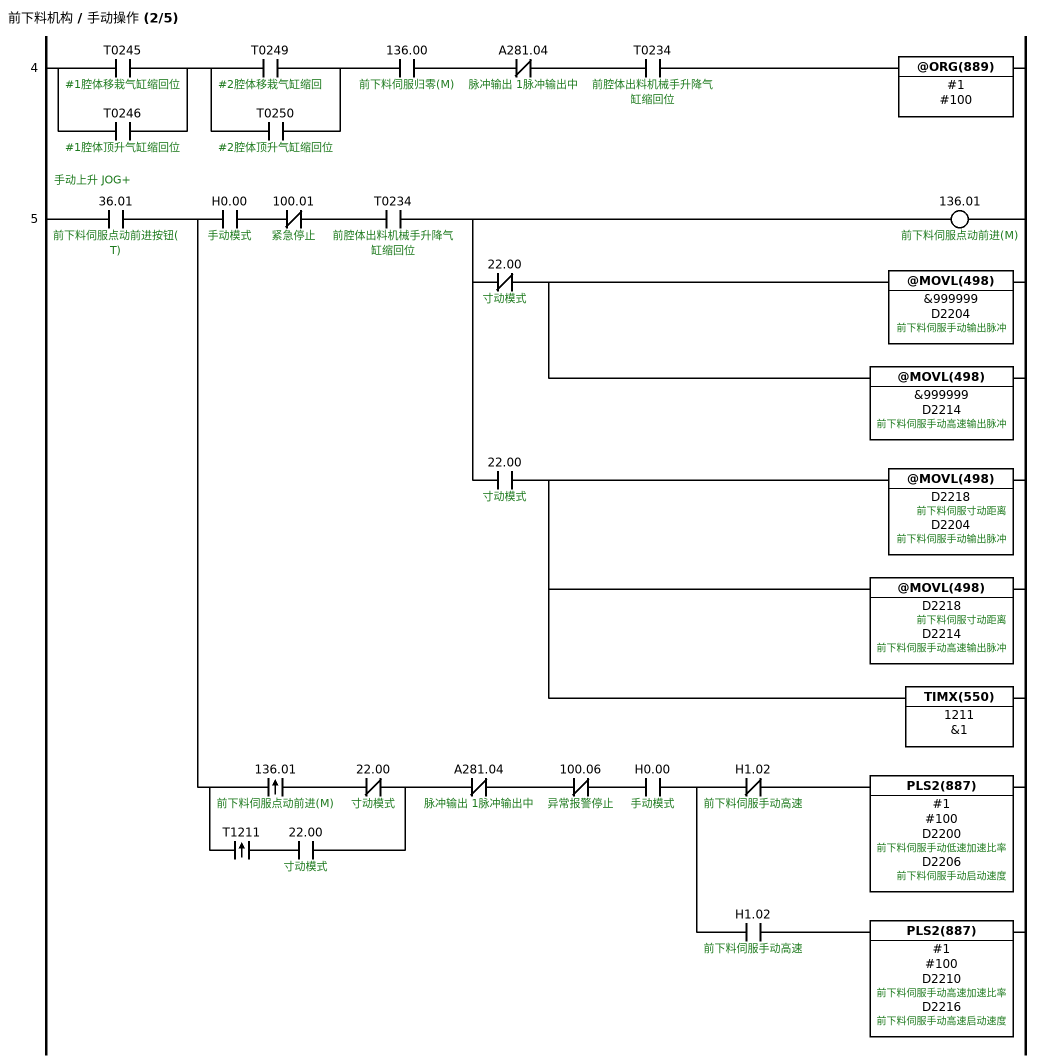
; rung 4
LD T0245  ; #1腔体移栽气缸缩回位
OR T0246  ; #1腔体顶升气缸缩回位
LD T0249  ; #2腔体移栽气缸缩回
OR T0250  ; #2腔体顶升气缸缩回位
ANDLD
AND 136.00  ; 前下料伺服归零(M)
ANDNOT A281.04  ; 脉冲输出 1脉冲输出中
AND T0234  ; 前腔体出料机械手升降气缸缩回位
@ORG(889) #1 #100
; rung 5: 手动上升 JOG+
LD 36.01  ; 前下料伺服点动前进按钮(T)
OUT TR0
AND H0.00  ; 手动模式
ANDNOT 100.01  ; 紧急停止
AND T0234  ; 前腔体出料机械手升降气缸缩回位
OUT TR1
OUT 136.01  ; 前下料伺服点动前进(M)
ANDNOT 22.00  ; 寸动模式
@MOVL(498) &999999 D2204  ; 前下料伺服手动输出脉冲
@MOVL(498) &999999 D2214  ; 前下料伺服手动高速输出脉冲
LD TR1
AND 22.00  ; 寸动模式
@MOVL(498) D2218 D2204  ; 前下料伺服寸动距离, 前下料伺服手动输出脉冲
@MOVL(498) D2218 D2214  ; 前下料伺服寸动距离, 前下料伺服手动高速输出脉冲
TIMX(550) 1211 &1
LD TR0
@LD 136.01  ; 前下料伺服点动前进(M)
ANDNOT 22.00  ; 寸动模式
@LD T1211
AND 22.00  ; 寸动模式
ORLD
ANDLD
ANDNOT A281.04  ; 脉冲输出 1脉冲输出中
ANDNOT 100.06  ; 异常报警停止
AND H0.00  ; 手动模式
OUT TR0
ANDNOT H1.02  ; 前下料伺服手动高速
PLS2(887) #1 #100 D2200 D2206  ; 前下料伺服手动低速加速比率, 前下料伺服手动启动速度
LD TR0
AND H1.02  ; 前下料伺服手动高速
PLS2(887) #1 #100 D2210 D2216  ; 前下料伺服手动高速加速比率, 前下料伺服手动高速启动速度

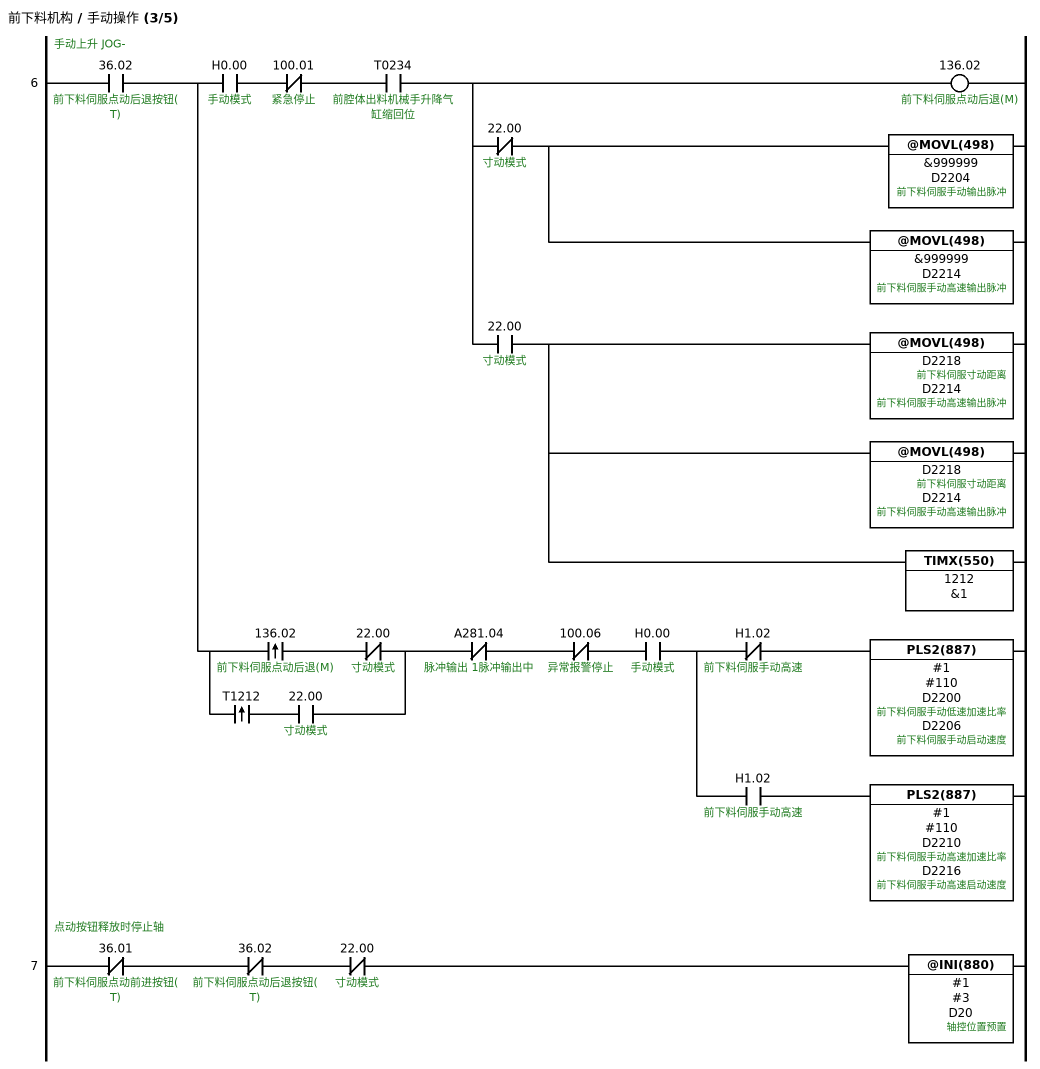
; rung 6: 手动上升 JOG-
LD 36.02  ; 前下料伺服点动后退按钮(T)
OUT TR0
AND H0.00  ; 手动模式
ANDNOT 100.01  ; 紧急停止
AND T0234  ; 前腔体出料机械手升降气缸缩回位
OUT TR1
OUT 136.02  ; 前下料伺服点动后退(M)
ANDNOT 22.00  ; 寸动模式
@MOVL(498) &999999 D2204  ; 前下料伺服手动输出脉冲
@MOVL(498) &999999 D2214  ; 前下料伺服手动高速输出脉冲
LD TR1
AND 22.00  ; 寸动模式
@MOVL(498) D2218 D2214  ; 前下料伺服寸动距离, 前下料伺服手动高速输出脉冲
@MOVL(498) D2218 D2214  ; 前下料伺服寸动距离, 前下料伺服手动高速输出脉冲
TIMX(550) 1212 &1
LD TR0
@LD 136.02  ; 前下料伺服点动后退(M)
ANDNOT 22.00  ; 寸动模式
@LD T1212
AND 22.00  ; 寸动模式
ORLD
ANDLD
ANDNOT A281.04  ; 脉冲输出 1脉冲输出中
ANDNOT 100.06  ; 异常报警停止
AND H0.00  ; 手动模式
OUT TR0
ANDNOT H1.02  ; 前下料伺服手动高速
PLS2(887) #1 #110 D2200 D2206  ; 前下料伺服手动低速加速比率, 前下料伺服手动启动速度
LD TR0
AND H1.02  ; 前下料伺服手动高速
PLS2(887) #1 #110 D2210 D2216  ; 前下料伺服手动高速加速比率, 前下料伺服手动高速启动速度
; rung 7: 点动按钮释放时停止轴
LDNOT 36.01  ; 前下料伺服点动前进按钮(T)
ANDNOT 36.02  ; 前下料伺服点动后退按钮(T)
ANDNOT 22.00  ; 寸动模式
@INI(880) #1 #3 D20  ; 轴控位置预置

